			// Không blend tại bước chuyển hệ tọa độ.
			MotionBlendRadius := 0.0;
	
			// Motion chạy trong Robot Base/MCS.
			MotionCoordSystem := E_AppCoordSystem.APP_COORD_ROBOT_BASE;
	
			// MoveL.
			MotionCommand := 2;
	
			// Phát yêu cầu tới Motion Adapter.
			xMotionRequestPending := TRUE;
			xMotionIssued := TRUE;
	
		END_IF;
	
		// Motion Adapter đã nhận lệnh.
		IF MotionAccepted AND xMotionRequestPending THEN
			xMotionRequestPending := FALSE;
			xMotionActive := TRUE;
		END_IF;
	
		// Điểm Safe Leave hoàn thành.
		IF MotionDone AND xMotionActive THEN
	
			xMotionActive := FALSE;
			xMotionIssued := FALSE;
			xMotionRequestPending := FALSE;
	
			Runtime.State := E_TrackingState.TRK_MOVE_PLACE;
	
		// Motion Safe Leave báo lỗi.
		ELSIF MotionError AND xMotionActive THEN
	
			xMotionActive := FALSE;
			xMotionIssued := FALSE;
			xMotionRequestPending := FALSE;
	
			Runtime.Response.Error := TRUE;
			Runtime.Response.ErrorID := MotionErrorID;
	
			Runtime.State := E_TrackingState.TRK_ERROR;
	
		END_IF;
		

    //=========================================================================
    // TRK_MOVE_PLACE
    // Di chuyển từ LeavePos tới PlacePos trong hệ robot/base.
    //=========================================================================
    E_TrackingState.TRK_MOVE_PLACE:

        // Giữ hút tới khi tới điểm đặt.
        VacuumCommand := xVacuumCaptured;

        // Tạo request Place mới.
        IF NOT xMotionIssued AND NOT xMotionRequestPending AND NOT xMotionActive THEN

            // Gán điểm Place.
            MotionTarget := Config.PlacePos;

            // Gán tốc độ Place.
            MotionSpeed := Config.Motion.Place.Speed;

            // Gán gia tốc Place.
            MotionAcceleration := Config.Motion.Place.Acceleration;

            // Gán giảm tốc Place.
            MotionDeceleration := Config.Motion.Place.Deceleration;

            // Gán jerk Place.
            MotionJerk := Config.Motion.Place.Jerk;

            // Gán blend Place.
            MotionBlendRadius := Config.Motion.Place.BlendRadius;

            // Place chạy trong hệ robot/base.
            MotionCoordSystem := E_AppCoordSystem.APP_COORD_ROBOT_BASE;

            // Mã lệnh MoveL.
            MotionCommand := 2;

            // Bật request pending.
            xMotionRequestPending := TRUE;

            // Đánh dấu đã tạo lệnh.
            xMotionIssued := TRUE;
        END_IF;

        // Adapter đã nhận request.
        IF MotionAccepted AND xMotionRequestPending THEN
            xMotionRequestPending := FALSE;
            xMotionActive := TRUE;
        END_IF;

        // Place hoàn thành.
        IF MotionDone AND xMotionActive THEN
            xMotionActive := FALSE;
            xMotionIssued := FALSE;

            Runtime.State := E_TrackingState.TRK_RELEASE_PRODUCT;

        // Place lỗi.
        ELSIF MotionError AND xMotionActive THEN
            xMotionActive := FALSE;

            Runtime.Response.Error := TRUE;
            Runtime.Response.ErrorID := MotionErrorID;

            Runtime.State := E_TrackingState.TRK_ERROR;
        END_IF;

    //=========================================================================
    // TRK_RELEASE_PRODUCT
    // Tắt hút, bật thổi và chuẩn bị timer.
    //=========================================================================
    E_TrackingState.TRK_RELEASE_PRODUCT:

        // Tắt hút để nhả sản phẩm.
        VacuumCommand := FALSE;

        // Bật van thổi.
        BlowCommand := TRUE;

        // Reset timer thổi trước khi vào state chờ.
        tonBlow(IN := FALSE);

        // Chuyển sang chờ đủ thời gian thổi.
        Runtime.State := E_TrackingState.TRK_WAIT_BLOW;

    //=========================================================================
    // TRK_WAIT_BLOW
    // Giữ thổi trong Config.BlowTime.
    //=========================================================================
    E_TrackingState.TRK_WAIT_BLOW:

        // Bảo đảm hút tắt.
        VacuumCommand := FALSE;

        // Giữ van thổi bật.
        BlowCommand := TRUE;

        // Chạy timer thổi.
        tonBlow(
            IN := TRUE,
            PT := Config.BlowTime
        );

        // Khi hết thời gian thổi.
        IF tonBlow.Q THEN
            // Reset timer.
            tonBlow(IN := FALSE);

            // Tắt thổi.
            BlowCommand := FALSE;

            // Đánh dấu object đã PICKED.
            Queue.Objects[Runtime.SelectedObjectIndex].State := E_TrackingObjectState.OBJ_PICKED;

            // Giải phóng cờ Reserved.
            Queue.Objects[Runtime.SelectedObjectIndex].Reserved := FALSE;

            // Giải phóng ActiveIndex.
            Queue.ActiveIndex := GVL.C_INVALID_INDEX;

            // Báo gắp thành công.
            Runtime.PickSuccess := TRUE;

            // Xóa object active trong Runtime.
            Runtime.SelectedObjectIndex := 0;
            Runtime.SelectedObjectID := 0;

            // Xóa trạng thái đã giữ vật.
            xVacuumCaptured := FALSE;

            // Phát Done.
            Runtime.Response.Done := TRUE;

            // Chuyển sang Complete.
            Runtime.State := E_TrackingState.TRK_COMPLETE;
        END_IF;

    //=========================================================================
    // TRK_COMPLETE
    // Kết thúc một object; nếu Execute còn TRUE thì tìm object tiếp theo.
    //=========================================================================
    E_TrackingState.TRK_COMPLETE:

        // Chu trình một object đã hoàn thành.
		Runtime.Response.Busy := FALSE;
		Runtime.Response.Done := TRUE;
	
		// Giữ output ở trạng thái an toàn.
		VacuumCommand := FALSE;
		BlowCommand := FALSE;
	
		// Chỉ về IDLE khi tầng Command Engine hạ Execute.
		IF NOT Execute THEN
			Runtime.Response.Accepted := FALSE;
			Runtime.Response.Done := FALSE;
			Runtime.State := E_TrackingState.TRK_IDLE;
		END_IF;


    //=========================================================================
    // TRK_ABORT_ACTIVE
    // Hủy motion vì object vượt vùng trước khi VacuumOK.
    //=========================================================================
    E_TrackingState.TRK_ABORT_ACTIVE:

        // Tắt hút vì chưa giữ được vật.
        VacuumCommand := FALSE;

        // Tắt thổi.
        BlowCommand := FALSE;

        // Bật yêu cầu abort motion.
        MotionAbort := TRUE;

        // Khi Motion Manager xác nhận abort hoàn tất.
        IF MotionAbortDone THEN
            // Hạ yêu cầu abort.
            MotionAbort := FALSE;

            // Xóa trạng thái motion.
            xMotionIssued := FALSE;
            xMotionRequestPending := FALSE;
            xMotionActive := FALSE;

            // Nếu PCS không còn InUse thì có thể tắt tracking.
            IF NOT fbTrackBelt.InUse THEN
                xTrackExecute := FALSE;

                // Chuyển sang vị trí an toàn.
                Runtime.State := E_TrackingState.TRK_MOVE_SAFE;
            END_IF;
        END_IF;

    //=========================================================================
    // TRK_MOVE_SAFE
    // Đưa robot về LeavePos sau khi bỏ object.
    //=========================================================================
    E_TrackingState.TRK_MOVE_SAFE:

        // Tắt hút.
        VacuumCommand := FALSE;

        // Tạo request Move Safe.
        IF NOT xMotionIssued AND NOT xMotionRequestPending AND NOT xMotionActive THEN

            // Dùng LeavePos làm điểm an toàn.
            MotionTarget := Config.LeavePos;

            // Dùng thông số Leave.
            MotionSpeed := Config.Motion.Leave.Speed;

            MotionAcceleration := Config.Motion.Leave.Acceleration;

            MotionDeceleration := Config.Motion.Leave.Deceleration;

            MotionJerk := Config.Motion.Leave.Jerk;

            MotionBlendRadius := Config.Motion.Leave.BlendRadius;

            // Chạy trong hệ robot/base.
            MotionCoordSystem := E_AppCoordSystem.APP_COORD_ROBOT_BASE;

            // Mã lệnh MoveL.
            MotionCommand := 2;

            // Bật request pending.
            xMotionRequestPending := TRUE;

            // Đánh dấu đã tạo lệnh.
            xMotionIssued := TRUE;
        END_IF;

        // Adapter đã nhận request.
        IF MotionAccepted AND xMotionRequestPending THEN
            xMotionRequestPending := FALSE;
            xMotionActive := TRUE;
        END_IF;

        // Move Safe hoàn thành.
        IF MotionDone AND xMotionActive THEN
            xMotionActive := FALSE;
            xMotionIssued := FALSE;

            Runtime.State := E_TrackingState.TRK_RELEASE_OBJECT;

        // Move Safe lỗi.
        ELSIF MotionError AND xMotionActive THEN
            xMotionActive := FALSE;

            Runtime.Response.Error := TRUE;
            Runtime.Response.ErrorID := MotionErrorID;

            Runtime.State := E_TrackingState.TRK_ERROR;
        END_IF;

    //=========================================================================
    // TRK_RELEASE_OBJECT
    // Giải phóng object MISSED và tiếp tục object kế tiếp.
    //=========================================================================
    E_TrackingState.TRK_RELEASE_OBJECT:

        // Tắt hút.
        VacuumCommand := FALSE;

        // Chỉ release khi PCS không còn InUse.
        IF NOT fbTrackBelt.InUse THEN
            // Tắt tracking PCS.
            xTrackExecute := FALSE;

            // Kiểm tra index trước khi truy cập Queue.
            IF Runtime.SelectedObjectIndex >= 1 AND Runtime.SelectedObjectIndex <= GVL.C_MAX_TRACK_OBJECTS THEN

                // Giải phóng object.
                Queue.Objects[Runtime.SelectedObjectIndex].Reserved := FALSE;
            END_IF;

            // Giải phóng ActiveIndex.
            Queue.ActiveIndex := GVL.C_INVALID_INDEX;

            // Xóa object active trong Runtime.
            Runtime.SelectedObjectIndex := 0;
            Runtime.SelectedObjectID := 0;

            // Xóa thông tin PCS.
            Runtime.PCSInfo.Valid := FALSE;
            Runtime.PCSInfo.InUse := FALSE;

            // Xóa trạng thái tool.
            xVacuumCaptured := FALSE;

            // Xóa trạng thái motion.
            xMotionIssued := FALSE;
            xMotionRequestPending := FALSE;
            xMotionActive := FALSE;

            // Tiếp tục tìm object khác.
            Runtime.State := E_TrackingState.TRK_FIND_OBJECT;
        END_IF;

    //=========================================================================
    // TRK_ABORTING
    // Hủy toàn ứng dụng khi Execute bị hạ.
    //=========================================================================
    E_TrackingState.TRK_ABORTING:

        // Tắt hút.
        VacuumCommand := FALSE;

        // Tắt thổi.
        BlowCommand := FALSE;

        // Yêu cầu abort motion.
        MotionAbort := TRUE;

        // Nếu có object active thì đánh dấu ABORTED.
        IF Runtime.SelectedObjectIndex >= 1 AND Runtime.SelectedObjectIndex <= GVL.C_MAX_TRACK_OBJECTS THEN

            Queue.Objects[Runtime.SelectedObjectIndex].State := E_TrackingObjectState.OBJ_ABORTED;

            Queue.Objects[Runtime.SelectedObjectIndex].Reserved := FALSE;
        END_IF;

        // Khi abort motion xong và PCS không còn InUse.
        IF MotionAbortDone AND NOT fbTrackBelt.InUse THEN

            // Hạ abort.
            MotionAbort := FALSE;

            // Tắt tracking PCS.
            xTrackExecute := FALSE;

            // Giải phóng ActiveIndex.
            Queue.ActiveIndex := GVL.C_INVALID_INDEX;

            // Xóa object active.
            Runtime.SelectedObjectIndex := 0;
            Runtime.SelectedObjectID := 0;

            // Xóa Busy và Accepted.
            Runtime.Response.Busy := FALSE;
            Runtime.Response.Accepted := FALSE;

            // Về IDLE.
            Runtime.State := E_TrackingState.TRK_IDLE;
        END_IF;

    //=========================================================================
    // TRK_ERROR
    // Giữ lỗi để Application Manager/HMI đọc.
    //=========================================================================
    E_TrackingState.TRK_ERROR:

        // Manager không còn xử lý bình thường.
        Runtime.Response.Busy := FALSE;

        // Giữ cờ Error.
        Runtime.Response.Error := TRUE;

        // Tắt hút.
        VacuumCommand := FALSE;

        // Tắt thổi.
        BlowCommand := FALSE;

        // Yêu cầu abort motion.
        MotionAbort := TRUE;

        // Nếu có object active thì đánh dấu ERROR.
        IF Runtime.SelectedObjectIndex >= 1 AND Runtime.SelectedObjectIndex <= GVL.C_MAX_TRACK_OBJECTS THEN

            Queue.Objects[Runtime.SelectedObjectIndex].State := E_TrackingObjectState.OBJ_ERROR;

            Queue.Objects[Runtime.SelectedObjectIndex].Reserved := FALSE;
        END_IF;

        // Chỉ tắt tracking khi PCS không còn InUse.
        IF NOT fbTrackBelt.InUse THEN
            xTrackExecute := FALSE;
        END_IF;

    //=========================================================================
    // STATE KHÔNG HỢP LỆ
    //=========================================================================
    ELSE
        // Báo lỗi state không hợp lệ.
        Runtime.Response.Error := TRUE;

        // Mã lỗi nội bộ cho state không hợp lệ.
        Runtime.Response.ErrorID := 6999;

        // Chuyển về TRK_ERROR.
        Runtime.State := E_TrackingState.TRK_ERROR;

END_CASE;

END_FUNCTION_BLOCK

// Just_Motion_Control_x86_64_Linux_SM_WV/Application/FB_/ConveyorTrack/FB_TrackingMotionQueueAdapter_B
FUNCTION_BLOCK FB_TrackingMotionQueueAdapter_B
VAR_INPUT
    Enable : BOOL; // Biến nội bộ Enable.
    Reset : BOOL; // Biến nội bộ Reset.
    Request : BOOL; // Biến nội bộ Request.
    Abort : BOOL; // Biến nội bộ Abort.
    Target : ST_POS; // Biến nội bộ Target.
    Speed : REAL; // Biến nội bộ Speed.
    Acceleration : REAL; // Biến nội bộ Acceleration.
    Deceleration : REAL; // Biến nội bộ Deceleration.
    Jerk : REAL; // Biến nội bộ Jerk.
    BlendRadius : REAL; // Biến nội bộ BlendRadius.
    CoordSystem : E_AppCoordSystem; // Biến nội bộ CoordSystem.
    Command : UINT; // Biến nội bộ Command.
    LogicSimulation : BOOL; // Logic-only simulation không push vào robot.
    LogicMotionDuration : TIME := TIME#300ms; // Biến nội bộ LogicMotionDuration.
END_VAR

VAR_OUTPUT
    Accepted : BOOL; // Biến nội bộ Accepted.
    Busy : BOOL; // Biến nội bộ Busy.
    Done : BOOL; // Biến nội bộ Done.
    Error : BOOL; // Biến nội bộ Error.
    ErrorID : UDINT; // Biến nội bộ ErrorID.
    AbortDone : BOOL; // Biến nội bộ AbortDone.
END_VAR

VAR
    fbPush : FB_MotionQueuePush_B; // Biến nội bộ fbPush.
    rtRequest : R_TRIG; // Biến nội bộ rtRequest.
    tonLogicMotion : TON; // Biến nội bộ tonLogicMotion.
    stItem : ST_MotionQueueItem; // Biến nội bộ stItem.
    xPushExecute : BOOL; // Biến nội bộ xPushExecute.
    xWaitingMotionResult : BOOL; // Biến nội bộ xWaitingMotionResult.
    xAcceptedLatched : BOOL; // Biến nội bộ xAcceptedLatched.
    diRequestSequence : DINT := -1000; // Biến nội bộ diRequestSequence.
    iActiveSourceStep : INT; // Biến nội bộ iActiveSourceStep.
END_VAR

Accepted := FALSE;
Done := FALSE;
AbortDone := FALSE;

// Error không nên giữ từ request cũ khi Adapter đang không chờ motion.
IF NOT xPushExecute AND NOT xWaitingMotionResult THEN
    Error := FALSE;
    ErrorID := 0;
END_IF;

// IF Reset OR NOT Enable THEN
//     xPushExecute := FALSE;
//     xWaitingMotionResult := FALSE;
//     xAcceptedLatched := FALSE;
//     Busy := FALSE;
//     Error := FALSE;
//     ErrorID := 0;
//     tonLogicMotion(IN := FALSE);
//     fbPush(Execute := FALSE, Item := stItem);
//     RETURN;
// END_IF;

IF Reset OR NOT Enable THEN

    // Hạ yêu cầu push vào Motion Queue.
    xPushExecute := FALSE;

    // Không còn chờ kết quả motion trước.
    xWaitingMotionResult := FALSE;

    // Xóa cờ Accepted nội bộ.
    xAcceptedLatched := FALSE;

    // Xóa trạng thái output.
    Accepted := FALSE;
    Busy := FALSE;
    Done := FALSE;
    Error := FALSE;
    ErrorID := 0;
    AbortDone := FALSE;

    // Xóa SourceStep của request cũ.
    iActiveSourceStep := 0;

    // Hạ yêu cầu Abort còn sót lại.
    GVL.B_MotionAbortReq := FALSE;

    // Reset timer mô phỏng.
    tonLogicMotion(IN := FALSE);

    // Reset FB Push Motion Queue.
    fbPush(Execute := FALSE, Item := stItem);

    RETURN;
END_IF;

IF Abort THEN
    IF LogicSimulation THEN
        xWaitingMotionResult := FALSE;
        Busy := FALSE;
        AbortDone := TRUE;
    ELSE
        GVL.B_MotionAbortReq := TRUE;
        IF GVL.B_MotionAbortDone THEN
            GVL.B_MotionAbortReq := FALSE;
            xWaitingMotionResult := FALSE;
            Busy := FALSE;
            AbortDone := TRUE;
        END_IF;
    END_IF;
    RETURN;
END_IF;

rtRequest(CLK := Request);

//=============================================================================
// LOGIC-ONLY SIMULATION
//=============================================================================
IF LogicSimulation THEN
    IF rtRequest.Q AND NOT Busy THEN
        Accepted := TRUE;
        Busy := TRUE;
        tonLogicMotion(IN := FALSE);
    END_IF;

    tonLogicMotion(IN := Busy, PT := LogicMotionDuration);

    IF tonLogicMotion.Q THEN
        tonLogicMotion(IN := FALSE);
        Busy := FALSE;
        Done := TRUE;
    END_IF;

    RETURN;
END_IF;

//=============================================================================
// ROBOT REAL: ĐÓNG GÓI VÀ PUSH VÀO MOTION QUEUE ROBOT B
//=============================================================================
IF rtRequest.Q AND NOT xPushExecute AND NOT xWaitingMotionResult THEN
    diRequestSequence := diRequestSequence - 1;
    IF diRequestSequence < -30000 THEN diRequestSequence := -1000; END_IF;
    iActiveSourceStep := DINT_TO_INT(diRequestSequence);

    stItem.Cmd := E_RobotCmd.CMD_MovL;
    stItem.SourceStep := iActiveSourceStep;
    stItem.PointNo := 0;
    stItem.MidPointNo := 0;
    stItem.EndPointNo := 0;
    stItem.Speed := REAL_TO_LREAL(Speed);
    stItem.BlendMode := GVL.C_TM_None;
    stItem.BlendRadius := REAL_TO_LREAL(BlendRadius);
    stItem.CircleMode := 0;
    stItem.PathChoice := 0;
    stItem.SkipPositionCheck := TRUE;

    stItem.UseDirectPosition := TRUE;
    stItem.DirectPosition := Target;
    stItem.DirectCoordSystem := F_MapAppCoordSystem(Coord := CoordSystem);
    stItem.Acceleration := REAL_TO_LREAL(Acceleration);
    stItem.Deceleration := REAL_TO_LREAL(Deceleration);
    stItem.Jerk := REAL_TO_LREAL(Jerk);
    stItem.ApplicationCommandID := TO_UDINT(ABS(iActiveSourceStep));

    xPushExecute := TRUE;
END_IF;

fbPush(Execute := xPushExecute, Item := stItem);

IF xPushExecute AND fbPush.Done THEN
    xPushExecute := FALSE;
    xWaitingMotionResult := TRUE;
    xAcceptedLatched := TRUE;
    Accepted := TRUE;
    Busy := TRUE;
END_IF;

IF xPushExecute AND fbPush.Error THEN
    xPushExecute := FALSE;
    Error := TRUE;
    ErrorID := 7201; // Motion Queue full / Push failed.
END_IF;

// Reset handshake của FB Push sau khi push xong.
IF NOT xPushExecute THEN fbPush(Execute := FALSE, Item := stItem); END_IF;

// Theo dõi đúng item bằng SourceStep âm riêng của Application.
IF xWaitingMotionResult THEN
    Busy := TRUE;

//     IF GVL.B_MotionDonePulse AND GVL.B_MotionDoneStep = iActiveSourceStep THEN
//         xWaitingMotionResult := FALSE;
//         Busy := FALSE;
//         Done := TRUE;
//     END_IF;
// 
//     IF GVL.B_MotionErrorPulse AND GVL.B_MotionErrorStep = iActiveSourceStep THEN
//         xWaitingMotionResult := FALSE;
//         Busy := FALSE;
//         Error := TRUE;
//         ErrorID := INT_TO_UDINT(GVL.B_MotionErrorCode);
//     END_IF;
	
	IF GVL.B_MotionDonePulse AND GVL.B_MotionDoneStep = iActiveSourceStep THEN
		xWaitingMotionResult := FALSE;
		xAcceptedLatched := FALSE;
		Busy := FALSE;
		Done := TRUE;
	END_IF;
	
	// Motion hiện tại báo lỗi đúng SourceStep.
	IF GVL.B_MotionErrorPulse AND GVL.B_MotionErrorStep = iActiveSourceStep THEN
		xWaitingMotionResult := FALSE;
		xAcceptedLatched := FALSE;
		Busy := FALSE;
		Error := TRUE;
		ErrorID := INT_TO_UDINT(GVL.B_MotionErrorCode);
	END_IF;
END_IF;

END_FUNCTION_BLOCK

// Just_Motion_Control_x86_64_Linux_SM_WV/Application/FB_/TOOL/FB_SelectRobotTool_B
FUNCTION_BLOCK FB_SelectRobotTool_B
VAR_INPUT
    Execute : BOOL; // Xung Execute.
    Reset : BOOL; // Reset FB.
    ToolID : UINT; // ToolID cần chọn.
END_VAR

VAR_OUTPUT
    Done : BOOL; // Tool đã được chọn.
    Busy : BOOL; // FB đang xử lý.
    Error : BOOL; // FB lỗi.
    ErrorID : UDINT; // Mã lỗi.
END_VAR

VAR
    rtExecute : R_TRIG; // Bắt cạnh Execute.
    fbGroupSetTool : SMC_GroupSetTool; // TODO: Khai báo instance SMC_GroupSetTool đúng theo version thư viện.
    xExecuteTool : BOOL; // Biến nội bộ xExecuteTool.
    udiMyRequestID : UDINT := 0; // RequestID thuộc transaction hiện tại.
END_VAR

//=============================================================================
// FB_SelectRobotTool
//-----------------------------------------------------------------------------
// ToolID = Number_Tool.
// Không gọi SMC_GroupSetTool tại đây.
// POU_COORDINATE_ là nơi duy nhất Apply TCP vào SCARA_B.
//=============================================================================

Done := FALSE;


//=============================================================================
// RESET
//=============================================================================
IF Reset THEN
    Busy := FALSE;
    Error := FALSE;
    ErrorID := 0;
    udiMyRequestID := 0;
    RETURN;
END_IF;


//=============================================================================
// DETECT EXECUTE
//=============================================================================
rtExecute(CLK := Execute);


//=============================================================================
// TẠO YÊU CẦU CHỌN / APPLY TOOL
//=============================================================================
IF rtExecute.Q AND NOT Busy THEN

    Busy := TRUE;
    Error := FALSE;
    ErrorID := 0;

    //---------------------------------------------------------------------
    // ToolID chính là Number_Tool.
    //
    // ToolID = 0 : No Tool Offset.
    // ToolID = 1 : Tool 1.
    // ToolID = 2 : Tool 2...
    //---------------------------------------------------------------------
    GVL.RB_B.Number_Tool := ToolID;

    //---------------------------------------------------------------------
    // Luôn tạo Request mới.
    // Nhờ vậy cùng ToolID nhưng TCP đã thay đổi vẫn được Apply lại.
    //---------------------------------------------------------------------
    GVL.g_udiRobotBToolApplyRequestB := GVL.g_udiRobotBToolApplyRequestB + 1;
    IF GVL.g_udiRobotBToolApplyRequestB = 0 THEN GVL.g_udiRobotBToolApplyRequestB := 1; END_IF;

    // Chốt Request của transaction này.
    udiMyRequestID := GVL.g_udiRobotBToolApplyRequestB;

END_IF;


//=============================================================================
// CHỜ KẾT QUẢ TỪ POU_COORDINATE_
//=============================================================================
IF Busy THEN

    //---------------------------------------------------------------------
    // APPLY ERROR
    //---------------------------------------------------------------------
    IF GVL.g_xRobotBToolApplyError THEN
        Busy := FALSE;
        Error := TRUE;
        ErrorID := GVL.g_udiRobotBToolApplyErrorID;

    //---------------------------------------------------------------------
    // APPLY DONE
    //---------------------------------------------------------------------
    ELSIF udiMyRequestID <> 0
    AND GVL.g_udiRobotBToolAppliedRequestB = udiMyRequestID THEN
        Busy := FALSE;
        Error := FALSE;
        ErrorID := 0;
        Done := TRUE;
    END_IF;

END_IF;





// (*
// ===============================================================================
// FUNCTION BLOCK
//     FB_SelectRobotTool
// 
// DESCRIPTION
//     Wrapper chọn Tool/TCP cho Robot.
// 
// TODO INTEGRATIONđ
//     Thay phần Logic-Only Placeholder bằng SMC_GroupSetTool đang có
//     trong project hiện tại.
// 
// EXPECTED FLOW
//     Execute rising edge
//         -> Call SMC_GroupSetTool
//         -> Wait Done/Error
//         -> Return Done/Error
// ===============================================================================
// *)
// 
// //=============================================================================
// // DEFAULT PULSE OUTPUT
// //=============================================================================
// Done := FALSE;
// 
// 
// //=============================================================================
// // RESET
// //=============================================================================
// IF Reset THEN
// 
//     Busy := FALSE;
// 
//     Error := FALSE;
//     ErrorID := 0;
// 
//     RETURN;
// 
// END_IF;
// 
// 
// //=============================================================================
// // DETECT EXECUTE
// //=============================================================================
// rtExecute(CLK := Execute);
// 
// 
// //=============================================================================
// // START TOOL SELECTION
// //=============================================================================
// IF rtExecute.Q AND NOT Busy THEN
// 
//     Busy := TRUE;
// 
//     Error := FALSE;
//     ErrorID := 0;
// 
// 
//     //=========================================================================
//     // TODO: CALL SMC_GROUPSETTOOL HERE
//     //-------------------------------------------------------------------------
//     // Ví dụ logic:
//     //
// 	fbGroupSetTool(
// 		Execute   := TRUE,
// 		AxisGroup := SCARA_B,
// 		ToolOffset := F_ConvertToolTCP(ToolTCP)
// 	);
// 	
// 	IF fbGroupSetTool.Done THEN
// 		Busy := FALSE;
// 		Done := TRUE;
// 	END_IF;
// 	
// 	IF fbGroupSetTool.Error THEN
// 		Busy := FALSE;
// 		Error := TRUE;
// 		ErrorID := fbGroupSetTool.ErrorID;
// 	END_IF;
//     //=========================================================================
// 
// 
// //     //-------------------------------------------------------------------------
// //     // LOGIC-ONLY PLACEHOLDER
// //     //-------------------------------------------------------------------------
// //     // Xóa hai dòng dưới sau khi nối SMC_GroupSetTool thực tế.
// //     Busy := FALSE;
// //     Done := TRUE;
// 
// END_IF;

END_FUNCTION_BLOCK

// Just_Motion_Control_x86_64_Linux_SM_WV/Application/FB_/TOOL/FB_ToolManager_B
FUNCTION_BLOCK FB_ToolManager_B
VAR_INPUT
    Enable : BOOL; // Cho phép Tool Manager.
    Command : ST_ToolCommand; // Command hiện tại.
    Config : ST_ToolConfig; // Cấu hình Tool.
END_VAR

VAR_IN_OUT
    Status : ST_ToolStatus; // Runtime Status của Tool.
END_VAR

VAR
    rtExecute : R_TRIG; // Bắt cạnh lên của Execute.
    eActiveCommand : E_ToolCommandType; // Lệnh Tool đang chạy.
    tonAction : TON; // Timer dùng khi không cấu hình DI.
    tonTimeout : TON; // Timer giới hạn thời gian lệnh Tool.
    tonConfirm : TON; // Timer xác nhận GripOK ổn định.
    xActionOK : BOOL; // Điều kiện lệnh Tool hoàn thành.
    xFeedbackDI : BOOL; // Giá trị DI đang kiểm tra.
    tAction : TIME; // Thời gian giả lập nếu không có Sensor.
    tTimeout : TIME; // Timeout của lệnh Tool.
END_VAR

(*
===============================================================================
FUNCTION BLOCK
    FB_ToolManager

DESCRIPTION
    Điều khiển một Tool độc lập.

SUPPORTED COMMANDS
    - DOWN
    - GRIP
    - UP
    - RELEASE

FEEDBACK RULE
    - Nếu DI Channel > 0:
          Dùng DI làm điều kiện hoàn thành.
    - Nếu DI Channel = 0:
          Dùng Timer cấu hình tương ứng.
    - Nếu UseUpDown = FALSE:
          DOWN và UP hoàn thành ngay.

IMPORTANT
    - Chỉ FB này được phép ghi request IO của Tool.
    - Interpreter không nên ghi trực tiếp vào các DO đã thuộc Tool.
===============================================================================
*)

//=============================================================================
// DEFAULT PULSE OUTPUTS
//=============================================================================
Status.Accepted := FALSE;
Status.Done := FALSE;


//=============================================================================
// COPY TOOL ID TO STATUS
//=============================================================================
Status.ToolID := Config.ToolID;


//=============================================================================
// RESET / DISABLE
//=============================================================================
IF NOT Enable OR Command.Reset THEN

    Status.Busy := FALSE;

    Status.Error := FALSE;
    Status.ErrorID := 0;

    Status.State :=
        E_ToolRuntimeState.IDLE;

    tonAction(IN := FALSE);
    tonTimeout(IN := FALSE);
    tonConfirm(IN := FALSE);

    RETURN;

END_IF;


//=============================================================================
// ABORT
//=============================================================================
IF Command.Abort THEN

    Status.Busy := FALSE;

    Status.Error := TRUE;
    Status.ErrorID := 9299;

    Status.State :=
        E_ToolRuntimeState.ERROR;

    RETURN;

END_IF;


//=============================================================================
// DETECT NEW COMMAND
//=============================================================================
rtExecute(CLK := Command.Execute);

IF rtExecute.Q AND NOT Status.Busy THEN

    // Lưu loại lệnh hiện tại.
    eActiveCommand :=
        Command.CommandType;

    // Handshake.
    Status.Accepted := TRUE;
    Status.Busy := TRUE;

    Status.Error := FALSE;
    Status.ErrorID := 0;

    Status.ResponseCommandID :=
        Command.CommandID;

    // Reset timer trước khi bắt đầu lệnh mới.
    tonAction(IN := FALSE);
    tonTimeout(IN := FALSE);
    tonConfirm(IN := FALSE);

    // Gán State runtime.
    CASE eActiveCommand OF

        E_ToolCommandType.DOWN:
            Status.State :=
                E_ToolRuntimeState.DOWNING;

        E_ToolCommandType.GRIP:
            Status.State :=
                E_ToolRuntimeState.GRIPPING;

        E_ToolCommandType.UP:
            Status.State :=
                E_ToolRuntimeState.UPPING;

        E_ToolCommandType.RELEASE:
            Status.State :=
                E_ToolRuntimeState.RELEASING;

        ELSE
            Status.Busy := FALSE;
            Status.Done := TRUE;

    END_CASE;

END_IF;


//=============================================================================
// NO ACTIVE COMMAND
//=============================================================================
IF NOT Status.Busy THEN
    RETURN;
END_IF;


//=============================================================================
// RESET LOCAL ACTION FLAGS
//=============================================================================
xActionOK := FALSE;
xFeedbackDI := FALSE;

tAction := T#0MS;
tTimeout := T#1S;


//=============================================================================
// EXECUTE ACTIVE COMMAND
//=============================================================================
CASE eActiveCommand OF


    //=========================================================================
    // ACTION: DOWN
    //=========================================================================
    E_ToolCommandType.DOWN:

        // Tool không có cơ cấu Up/Down.
        IF NOT Config.UseUpDown THEN

            xActionOK := TRUE;

        ELSE

            //-----------------------------------------------------------------
            // COMMAND DOWN OUTPUT
            //-----------------------------------------------------------------
			
			IF Config.IO.UseSingleUpDownDO THEN
				// Single DO: phat muc DOWN.
				IF Config.IO.UpDownDOChannel > 0 AND Config.IO.UpDownDOChannel <= GVL.C_MAX_DO THEN
					GVL.Y[Config.IO.UpDownDOChannel] := Config.IO.DownDOActiveLevel;
				END_IF;
			ELSE
				// Dual DO: bat Down, tat Up.
				IF Config.IO.DownDOChannel > 0 AND Config.IO.DownDOChannel <= GVL.C_MAX_DO THEN
					GVL.Y[Config.IO.DownDOChannel] := Config.IO.DownDOActiveLevel;
				END_IF;
			
				IF Config.IO.UpDOChannel > 0 AND Config.IO.UpDOChannel <= GVL.C_MAX_DO THEN
					GVL.Y[Config.IO.UpDOChannel] := NOT Config.IO.UpDOActiveLevel;
				END_IF;
			END_IF;


            //-----------------------------------------------------------------
            // CHECK DOWN FEEDBACK
            //-----------------------------------------------------------------
            IF Config.IO.DownOKDIChannel = 0 THEN

                // Không có DI -> dùng Timer.
                tAction :=
                    Config.DownTimeNoSensor;

                tonAction(
                    IN := TRUE,
                    PT := tAction
                );

                xActionOK :=
                    tonAction.Q;

            ELSE

                // Có DI -> dùng Sensor.
                xActionOK :=
                    GVL.X[
                        Config.IO.DownOKDIChannel
                    ] = Config.IO.DownOKDIActiveLevel;

            END_IF;


            // Timeout của DOWN.
            tTimeout :=
                Config.DownTimeout;

        END_IF;


    //=========================================================================
    // ACTION: GRIP
    //=========================================================================
    E_ToolCommandType.GRIP:

        //---------------------------------------------------------------------
        // RESET RELEASE OUTPUT
        //---------------------------------------------------------------------
        IF Config.IO.UseSingleGripReleaseDO THEN
			IF Config.IO.GripReleaseDOChannel > 0 AND Config.IO.GripReleaseDOChannel <= GVL.C_MAX_DO THEN
				GVL.Y[Config.IO.GripReleaseDOChannel] := Config.IO.GripDOActiveLevel;
			END_IF;
		ELSE
			IF Config.IO.ReleaseDOChannel > 0 AND Config.IO.ReleaseDOChannel <= GVL.C_MAX_DO THEN
				GVL.Y[Config.IO.ReleaseDOChannel] := NOT Config.IO.ReleaseDOActiveLevel;
			END_IF;
			IF Config.IO.GripDOChannel > 0 AND Config.IO.GripDOChannel <= GVL.C_MAX_DO THEN
				GVL.Y[Config.IO.GripDOChannel] := Config.IO.GripDOActiveLevel;
			END_IF;
		END_IF;


        //---------------------------------------------------------------------
        // CHECK GRIP FEEDBACK
        //---------------------------------------------------------------------
        IF Config.IO.GripOKDIChannel = 0 THEN

            // Không có GripOK DI -> dùng Timer.
            tAction :=
                Config.GripTimeNoSensor;

            tonAction(
                IN := TRUE,
                PT := tAction
            );

            xActionOK :=
                tonAction.Q;

        ELSE

            // Có GripOK DI.
            xFeedbackDI :=
                GVL.X[
                    Config.IO.GripOKDIChannel
                ] = Config.IO.GripOKDIActiveLevel;

            // Xác nhận tín hiệu ổn định.
            tonConfirm(
                IN := xFeedbackDI,
                PT := Config.GripConfirmDelay
            );

            xActionOK :=
                tonConfirm.Q;

        END_IF;


        // Timeout của GRIP.
        tTimeout :=
            Config.GripTimeout;


    //=========================================================================
    // ACTION: UP
    //=========================================================================
    E_ToolCommandType.UP:

        // Tool không có cơ cấu Up/Down.
        IF NOT Config.UseUpDown THEN

            xActionOK := TRUE;

        ELSE

            //-----------------------------------------------------------------
            // RESET DOWN OUTPUT
            //-----------------------------------------------------------------
			IF Config.IO.UseSingleUpDownDO THEN
				// Single DO: UP = dao muc DOWN.
				IF Config.IO.UpDownDOChannel > 0 AND Config.IO.UpDownDOChannel <= GVL.C_MAX_DO THEN
					GVL.Y[Config.IO.UpDownDOChannel] := NOT Config.IO.DownDOActiveLevel;
				END_IF;
			ELSE
				// Dual DO: tat Down, bat Up.
				IF Config.IO.DownDOChannel > 0 AND Config.IO.DownDOChannel <= GVL.C_MAX_DO THEN
					GVL.Y[Config.IO.DownDOChannel] := NOT Config.IO.DownDOActiveLevel;
				END_IF;
			
				IF Config.IO.UpDOChannel > 0 AND Config.IO.UpDOChannel <= GVL.C_MAX_DO THEN
					GVL.Y[Config.IO.UpDOChannel] := Config.IO.UpDOActiveLevel;
				END_IF;
			END_IF;


            //-----------------------------------------------------------------
            // CHECK UP FEEDBACK
            //-----------------------------------------------------------------
            IF Config.IO.UpOKDIChannel = 0 THEN

                // Không có DI -> dùng Timer.
                tAction :=
                    Config.UpTimeNoSensor;

                tonAction(
                    IN := TRUE,
                    PT := tAction
                );

                xActionOK :=
                    tonAction.Q;

            ELSE

                // Có DI -> dùng Sensor.
                xActionOK :=
                    GVL.X[
                        Config.IO.UpOKDIChannel
                    ] = Config.IO.UpOKDIActiveLevel;

            END_IF;


            // Timeout của UP.
            tTimeout :=
                Config.UpTimeout;

        END_IF;


    //=========================================================================
    // ACTION: RELEASE
    //=========================================================================
    E_ToolCommandType.RELEASE:

        //---------------------------------------------------------------------
        // RESET GRIP OUTPUT
        //---------------------------------------------------------------------
        IF Config.IO.UseSingleGripReleaseDO THEN
			IF Config.IO.GripReleaseDOChannel > 0 AND Config.IO.GripReleaseDOChannel <= GVL.C_MAX_DO THEN
				GVL.Y[Config.IO.GripReleaseDOChannel] := NOT Config.IO.GripDOActiveLevel;
			END_IF;
		ELSE
			IF Config.IO.GripDOChannel > 0 AND Config.IO.GripDOChannel <= GVL.C_MAX_DO THEN
				GVL.Y[Config.IO.GripDOChannel] := NOT Config.IO.GripDOActiveLevel;
			END_IF;
			IF Config.IO.ReleaseDOChannel > 0 AND Config.IO.ReleaseDOChannel <= GVL.C_MAX_DO THEN
				GVL.Y[Config.IO.ReleaseDOChannel] := Config.IO.ReleaseDOActiveLevel;
			END_IF;
		END_IF;


        //---------------------------------------------------------------------
        // RELEASE CURRENTLY USES TIMER
        //---------------------------------------------------------------------
        tAction :=
            Config.ReleaseTimeNoSensor;

        tonAction(
            IN := TRUE,
            PT := tAction
        );

        xActionOK :=
            tonAction.Q;


        // Timeout của RELEASE.
        tTimeout :=
            Config.ReleaseTimeout;

END_CASE;


//=============================================================================
// ACTION TIMEOUT
//=============================================================================
tonTimeout(
    IN := TRUE,
    PT := tTimeout
);


//=============================================================================
// COMMAND COMPLETE
//=============================================================================
IF xActionOK THEN

    // Reset timer.
    tonAction(IN := FALSE);
    tonTimeout(IN := FALSE);
    tonConfirm(IN := FALSE);

    // Hoàn thành Handshake.
    Status.Busy := FALSE;
    Status.Done := TRUE;

    Status.Error := FALSE;
    Status.ErrorID := 0;


    //-------------------------------------------------------------------------
    // UPDATE TOOL RUNTIME STATE
    //-------------------------------------------------------------------------
    CASE eActiveCommand OF

        E_ToolCommandType.DOWN:

            Status.State :=
                E_ToolRuntimeState.DOWN;


        E_ToolCommandType.GRIP:

            Status.State :=
                E_ToolRuntimeState.OCCUPIED;

            Status.Occupied :=
                TRUE;

            Status.HeldObjectID :=
                Command.ObjectID;

            Status.GripOK :=
                TRUE;


        E_ToolCommandType.UP:

            IF Status.Occupied THEN

                Status.State :=
                    E_ToolRuntimeState.OCCUPIED;

            ELSE

                Status.State :=
                    E_ToolRuntimeState.UP;

            END_IF;


        E_ToolCommandType.RELEASE:

            Status.State :=
                E_ToolRuntimeState.IDLE;

            Status.Occupied :=
                FALSE;

            Status.HeldObjectID :=
                0;

            Status.GripOK :=
                FALSE;

    END_CASE;


//=============================================================================
// COMMAND ERROR
//=============================================================================
ELSIF tonTimeout.Q THEN

    Status.Busy := FALSE;

    Status.Error := TRUE;

    // Mã lỗi được tạo từ loại lệnh Tool.
    Status.ErrorID :=
        9200 + TO_UDINT(eActiveCommand);

    Status.State :=
        E_ToolRuntimeState.ERROR;

END_IF;

END_FUNCTION_BLOCK

// Just_Motion_Control_x86_64_Linux_SM_WV/Application/PRG_MACHINE/POU_MODBUS
PROGRAM POU_MODBUS
VAR
	
	Modbus_TCP_slave_0: JMCMB.modbusTCPslaveINI;
	slaveRegisters_0: JMCMB.slaveRegisters;
	DATA : ARRAY[0..2000] OF INT;
	id, id2, id3 : INT;
	
	Modbus_TCP_slave_1: JMCMB.modbusTCPslaveINI;
	slaveRegisters_1: JMCMB.slaveRegisters;
	DATA1 : ARRAY[0..2000] OF INT;
	uiCamera : UINT;
	iCameraBase : INT;
	Enable_Modbus_Camera : ARRAY[0..GVL.C_MAX_VISION_CHANNELS] OF BOOL;
END_VAR

ACT_TCP_Sever();
//ACT_modbus();

ACTION ACT_TCP_Sever:
Modbus_TCP_slave_0(en := TRUE,
					iniID := 1,
					port	:= 1010,
					TCP_UDP	:= 	0,
					DelayRespTime := 300,
					connected =>,
					errID =>,
					Info	=>,
					errTotal =>);
slaveRegisters_0(	iniID := 1,
					modeTCP_RTU := 0,
					startAddr := 0,
					total		:= 2000,
					trans_data	:= DATA,
					errId =>,
					Info	=>,
					CMDTimes	=>);
					

//Enable_Modbus_Camera[1] := TRUE;
FOR uiCamera := 1 TO GVL.C_MAX_VISION_CHANNELS DO
	IF (GVL.g_aVisionConfig[uiCamera].Enable) THEN
		iCameraBase := (UINT_TO_INT(uiCamera) - 1) * 300;
	
		// Robot -> Vision: chỉ ghi 100 register đầu của Camera.
		FOR id := 0 TO 99 DO
			DATA[iCameraBase + id] := TO_INT(GVL.MODBUS[iCameraBase + id]);
		END_FOR;
	
		// Vision -> Robot: chỉ đọc 200 register sau của Camera.
		FOR id2 := 100 TO 299 DO
			GVL.MODBUS[iCameraBase + id2] := TO_WORD(DATA[iCameraBase + id2]);
		END_FOR;
	END_IF;
END_FOR;

// User Modbus
FOR id := 1200 TO 1599 DO
	DATA[id] := TO_INT(GVL.MODBUS[id]);
END_FOR;

// Vision -> Robot: chỉ đọc 200 register sau của Camera.
FOR id2 := 1600 TO 1999 DO
	GVL.MODBUS[id2] := TO_WORD(DATA[id2]);
END_FOR;

// iCameraBase := 0;
// 	
// // Robot -> Vision: chỉ ghi 100 register đầu của Camera.
// FOR id := 0 TO 99 DO
// 	DATA[iCameraBase + id] := TO_INT(GVL.MODBUS[iCameraBase + id]);
// END_FOR;
// 
// // Vision -> Robot: chỉ đọc 200 register sau của Camera.
// FOR id2 := 100 TO 299 DO
// 	GVL.MODBUS[iCameraBase + id2] := TO_WORD(DATA[iCameraBase + id2]);
// END_FOR;
// 
// FOR id3 := 1500 TO 1999 DO
// 	GVL.MODBUS[id3] := TO_WORD(DATA[id3]);   // luôn cập nhật
// END_FOR;


Modbus_TCP_slave_1(en := FALSE,
					iniID := 2,
					port	:= 1012,
					TCP_UDP	:= 	0,
					DelayRespTime := 300,
					connected =>,
					errID =>,
					Info	=>,
					errTotal =>);
slaveRegisters_1(	iniID := 2,
					modeTCP_RTU := 0,
					startAddr := 0,
					total		:= 2000,
					trans_data	:= DATA1,
					errId =>,
					Info	=>,
					CMDTimes	=>);
END_ACTION

END_PROGRAM

// Just_Motion_Control_x86_64_Linux_SM_WV/Application/PRG_MACHINE/PRG_VisionConfigInit
PROGRAM PRG_VisionConfigInit
VAR
    xInitialized : BOOL := FALSE;
END_VAR

//=============================================================================
// PRG_VisionConfigInit
//-----------------------------------------------------------------------------
// Khởi tạo cấu hình Vision một lần sau khi PLC RUN.
// Không ghi lặp mỗi scan để sau này HMI có thể sửa cấu hình.
//=============================================================================

IF NOT xInitialized THEN

    //=========================================================================
    // CAMERA 1
    //=========================================================================
    //GVL.g_aVisionConfig[1].Enable := TRUE;
    GVL.g_aVisionConfig[1].CameraID := 1;
    GVL.g_aVisionConfig[1].BaseAddress := 0;
    GVL.g_aVisionConfig[1].CommandOffset := 0;
    GVL.g_aVisionConfig[1].StatusOffset := 100;
    GVL.g_aVisionConfig[1].HeaderOffset := 101;
    GVL.g_aVisionConfig[1].DataOffset := 116;

    // Scale tạm dùng cho test.
    // Raw 10000 -> 10.000 mm.
    //GVL.g_aVisionConfig[1].PositionScale := 0.001;
    //GVL.g_aVisionConfig[1].AngleScale := 0.001;
    GVL.g_aVisionConfig[1].ScoreScale := 1.0;

//     GVL.g_aVisionConfig[1].TriggerTimeout := T#2S;
//     GVL.g_aVisionConfig[1].ResultTimeout := T#3S;
    GVL.g_aVisionConfig[1].BlockTimeout := T#1S;
//     GVL.g_aVisionConfig[1].MaxPointCount := 12;
    //GVL.g_aVisionConfig[1].MaxRetry := 2;

	
	//=============================================================================
	// VISION TRACKING SOURCE 1
	//-----------------------------------------------------------------------------
	// Nguồn Vision dùng để tạo Object cho Conveyor Tracking Robot A.
	// CameraID và JobID phải khớp Header của Result.
	//=============================================================================
	
// 	GVL.g_aVisionTrackingSourceConfigA[1].Enable := TRUE;
// 	GVL.g_aVisionTrackingSourceConfigA[1].VisionSourceID := 1;
// 	GVL.g_aVisionTrackingSourceConfigA[1].VisionSourceName := 'Vision Tracking Cam 1';
// 	
// 	GVL.g_aVisionTrackingSourceConfigA[1].CameraID := 1;
// 	GVL.g_aVisionTrackingSourceConfigA[1].JobID := 1;
// 	
// 	// Nếu Vision không trả ProductClassID thì dùng Class mặc định này.
// 	GVL.g_aVisionTrackingSourceConfigA[1].ProductClassID := 1;
// 	
// 	// Chỉ nhận Object đạt Score yêu cầu.
// 	GVL.g_aVisionTrackingSourceConfigA[1].MinimumScore := 70.0;
// 	GVL.g_aVisionTrackingSourceConfigA[1].MaxObjectCount := 10;
	
	//=============================================================================
	// SCALE
	//-----------------------------------------------------------------------------
	// Result Modbus Driver hiện đã decode X/Y/A ra engineering unit,
	// vì vậy ResultInPixel phải FALSE trong bài test hiện tại.
	//=============================================================================
// 	GVL.g_aVisionTrackingSourceConfigA[1].ResultInPixel := FALSE;
// 	GVL.g_aVisionTrackingSourceConfigA[1].MMPerPixelX := 1.0;
// 	GVL.g_aVisionTrackingSourceConfigA[1].MMPerPixelY := 1.0;
// 	
// 	//=============================================================================
// 	// VISION FINE OFFSET
// 	//=============================================================================
// 	GVL.g_aVisionTrackingSourceConfigA[1].VisionOffset.X := 0.0;
// 	GVL.g_aVisionTrackingSourceConfigA[1].VisionOffset.Y := 0.0;
// 	GVL.g_aVisionTrackingSourceConfigA[1].VisionOffset.Z := 0.0;
// 	GVL.g_aVisionTrackingSourceConfigA[1].VisionOffset.A := 0.0;
	
// 	//=============================================================================
// 	// DUPLICATE FILTER
// 	//=============================================================================
// 	GVL.g_aVisionTrackingSourceConfigA[1].DuplicateToleranceXMM := 10.0;
// 	GVL.g_aVisionTrackingSourceConfigA[1].DuplicateToleranceYMM := 10.0;
// 	GVL.g_aVisionTrackingSourceConfigA[1].DuplicateAngleDeg := 5.0;
	
	//=============================================================================
	// BACKGROUND TRIGGER
	//-----------------------------------------------------------------------------
	// Trong lúc test dữ liệu giả lập, chưa bật AutoTrigger để tránh sinh TriggerID mới.
	//=============================================================================
// 	GVL.g_aVisionTrackingSourceConfigA[1].AutoTrigger := FALSE;
// 	GVL.g_aVisionTrackingSourceConfigA[1].TriggerPitchMM := 50.0;
// 	GVL.g_aVisionTrackingSourceConfigA[1].TriggerOnlyWhenMoving := FALSE;
	GVL.g_aVisionTrackingSourceConfigA[1].MinimumTriggerVelocityMMs := 1.0;



    //=========================================================================
    // CAMERA 2
    //=========================================================================
    //GVL.g_aVisionConfig[2].Enable := FALSE;
    GVL.g_aVisionConfig[2].CameraID := 2;
    GVL.g_aVisionConfig[2].BaseAddress := 300;
    GVL.g_aVisionConfig[2].CommandOffset := 0;
    GVL.g_aVisionConfig[2].StatusOffset := 100;
    GVL.g_aVisionConfig[2].HeaderOffset := 101;
    GVL.g_aVisionConfig[2].DataOffset := 116;
    //GVL.g_aVisionConfig[2].PositionScale := 0.001;
    //GVL.g_aVisionConfig[2].AngleScale := 0.001;
    GVL.g_aVisionConfig[2].ScoreScale := 1.0;


    //=========================================================================
    // CAMERA 3
    //=========================================================================
    //GVL.g_aVisionConfig[3].Enable := FALSE;
    GVL.g_aVisionConfig[3].CameraID := 3;
    GVL.g_aVisionConfig[3].BaseAddress := 600;
    GVL.g_aVisionConfig[3].CommandOffset := 0;
    GVL.g_aVisionConfig[3].StatusOffset := 100;
    GVL.g_aVisionConfig[3].HeaderOffset := 101;
    GVL.g_aVisionConfig[3].DataOffset := 116;
    //GVL.g_aVisionConfig[3].PositionScale := 0.001;
    //GVL.g_aVisionConfig[3].AngleScale := 0.001;
    GVL.g_aVisionConfig[3].ScoreScale := 1.0;


    //=========================================================================
    // CAMERA 4
    //=========================================================================
    //GVL.g_aVisionConfig[4].Enable := FALSE;
    GVL.g_aVisionConfig[4].CameraID := 4;
    GVL.g_aVisionConfig[4].BaseAddress := 900;
    GVL.g_aVisionConfig[4].CommandOffset := 0;
    GVL.g_aVisionConfig[4].StatusOffset := 100;
    GVL.g_aVisionConfig[4].HeaderOffset := 101;
    GVL.g_aVisionConfig[4].DataOffset := 116;
    //GVL.g_aVisionConfig[4].PositionScale := 0.001;
    //GVL.g_aVisionConfig[4].AngleScale := 0.001;
    GVL.g_aVisionConfig[4].ScoreScale := 1.0;
	
	//=========================================================================
	// CAMERA 1
	//=========================================================================
	//GVL.g_aVisionConfig[1].Robot := E_VisionRobot.VIS_ROBOT_A;
	
	//=========================================================================
	// CAMERA 2
	//=========================================================================
	//GVL.g_aVisionConfig[2].Robot := E_VisionRobot.VIS_ROBOT_A;
	
	//=========================================================================
	// CAMERA 3
	//=========================================================================
	//GVL.g_aVisionConfig[3].Robot := E_VisionRobot.VIS_ROBOT_A;
	
	//=========================================================================
	// CAMERA 4
	//=========================================================================
	//GVL.g_aVisionConfig[4].Robot := E_VisionRobot.VIS_ROBOT_NONE;


    // Đánh dấu đã khởi tạo để không ghi lại mỗi scan.
    xInitialized := TRUE;

END_IF;

END_PROGRAM

// Just_Motion_Control_x86_64_Linux_SM_WV/Application/PRG_MACHINE/POU_CAM
PROGRAM POU_CAM
VAR
	RB_A_READ_CAM, RB_B_READ_CAM   	 : FB_Real_TO_Word_;
	RB_T1_WRITE, RB_T2_WRITE , RB_T1_READ_CAM_OFFSET , RB_T2_READ_CAM_OFFSET			 : FB_word_TO_real_;
	Connect_fail, bit_TRANS_modbus1, bit_RECEI_modbus1 : BOOL;
	TRIGGER_TOP, TRIGGER_DONE, Trigger_Busy : BOOL;
	R_Trig_TriggerDone : R_TRIG;
	T1,T2,T3,T4 : TON;
	i_Vs : INT;
	

END_VAR
VAR // added by the converter: edge detectors and wires of the graphical bodies
    _w1, _w2 : BOOL;
END_VAR

// // check Connect	
// bit_RECEI_modbus1 := GVL.MODBUS[100].0 OR GVL.MODBUS[100 + GVL.NB_Register_Modbus_VS *1].0 OR GVL.MODBUS[100 + GVL.NB_Register_Modbus_VS *2].0 OR GVL.MODBUS[100 + GVL.NB_Register_Modbus_VS *3].0;
// GVL.MODBUS[0].0 := bit_TRANS_modbus1;
// GVL.MODBUS[GVL.NB_Register_Modbus_VS *1].0 := bit_TRANS_modbus1;
// GVL.MODBUS[GVL.NB_Register_Modbus_VS *2].0 := bit_TRANS_modbus1;
// GVL.MODBUS[GVL.NB_Register_Modbus_VS *3].0 := bit_TRANS_modbus1;
// 
// /// Bit control Robot - VS
// i_Vs := 0;
// FOR i_Vs := 0 TO 2 BY 1 DO
// 	IF GVL.Data_Calib_RB[i_Vs].Use THEN
// 		// Tin hieu Trigger Modbus
// 		GVL.MODBUS[GVL.NB_Register_Modbus_VS *i_Vs].1 := GVL.Man_Calib_RB[i_Vs].Trigger_VS OR GVL.Auto_VS_RB[i_Vs].Trigger_VS;
// 		// Tin hieu bao Chay xong cac vi tri calib
// 		GVL.MODBUS[GVL.NB_Register_Modbus_VS *i_Vs].2 := GVL.Man_Calib_RB[i_Vs].Run_Pos_Calib_Done OR GVL.Auto_VS_RB[i_Vs].Run_Pos_Calib_Done;
// 		// Tin hieu bao Trigger Done tu VS System
// 		GVL.Man_Calib_RB[i_Vs].Trigger_Done := GVL.MODBUS[GVL.NB_Register_Modbus_VS *i_Vs + 100].1;
// 		GVL.Auto_VS_RB[i_Vs].Trigger_Done := GVL.MODBUS[GVL.NB_Register_Modbus_VS *i_Vs + 100].1;
// 		// Tin hieu bao Calib Done tu VS System
// 		GVL.Man_Calib_RB[i_Vs].Calib_VS_Done := GVL.MODBUS[GVL.NB_Register_Modbus_VS *i_Vs + 100].2;
// 		GVL.Auto_VS_RB[i_Vs].Calib_VS_Done := GVL.MODBUS[GVL.NB_Register_Modbus_VS *i_Vs + 100].2;		
// 	END_IF
// END_FOR
// // GVL.MODBUS[0].1 := TRIGGER_TOP;
// IF (GVL.MODBUS[0].1) THEN
// 	Trigger_Busy := TRUE;
// ELSE
// 	Trigger_Busy := FALSE;
// END_IF;
// //TRIGGER_DONE := GVL.MODBUS[100].1; // doc tin hieu bao trigger done
// // R_Trig_TriggerDone(CLK := GVL.MODBUS[100].1 );
// // IF Trigger_Busy AND R_Trig_TriggerDone.Q AND NOT GVL.X[8]  THEN
// // 	TRIGGER_DONE := TRUE;
// // END_IF
// 
// //TRIGGER_DONE := GVL.MODBUS[100].1;
// 
// GVL.Pro4_.Auto.Result_Trigger_Vs_Align_Done := TRIGGER_DONE;
// GVL.Pro4_.Man.Result_Trigger_Vs_Align_Done := TRIGGER_DONE;
// //  Bit control - Calib
// //GVL.MODBUS[0].2 := GVL.Pro4_.Man.Run_Calib_Pos_Done;
// GVL.Pro4_.Man.Result_Calib_Done := GVL.MODBUS[100].2;
// 
// 
// 
// // Funtion run
// ACT_TRIGGER_TOP();
// ACT_CHECKCONNECT();
// //ACT_Total();
// 
// 
// // 	RB_A_READ_CAM(	R_RB_X	:= TO_REAL(GVL.RB_A_.CUR_X),
// // 					R_RB_Y	:= TO_REAL(GVL.RB_A_.CUR_Y),
// // 					R_RB_r	:= TO_REAL(GVL.RB_A_.CUR_R),
// // 					LOW_RB_X	=> GVL.MODBUS[2],
// // 					HIGH_RB_X	=> GVL.MODBUS[3],
// // 					LOW_RB_Y	=> GVL.MODBUS[4],
// // 					HIGH_RB_Y	=> GVL.MODBUS[5],
// // 					LOW_RB_R	=> GVL.MODBUS[6],
// // 					HIGH_RB_R	=> GVL.MODBUS[7]);								
// // 	RB_B_READ_CAM(	R_RB_X	:= TO_REAL(GVL.RB_B_.CUR_X),
// // 					R_RB_Y	:= TO_REAL(GVL.RB_B_.CUR_Y),
// // 					R_RB_r	:= TO_REAL(GVL.RB_B_.CUR_R),
// // 					LOW_RB_X	=> GVL.MODBUS[8],
// // 					HIGH_RB_X	=> GVL.MODBUS[9],
// // 					LOW_RB_Y	=> GVL.MODBUS[10],
// // 					HIGH_RB_Y	=> GVL.MODBUS[11],
// // 					LOW_RB_R	=> GVL.MODBUS[12],
// // 					HIGH_RB_R	=> GVL.MODBUS[13]);	
// 								
// RB_T1_WRITE(W_LOW_CAM_X := GVL.MODBUS[102],
// 			W_HIGH_CAM_X := GVL.MODBUS[103],
// 			W_LOW_CAM_Y := GVL.MODBUS[104],
// 			W_HIGH_CAM_Y := GVL.MODBUS[105],
// 			W_LOW_CAM_R := GVL.MODBUS[106],
// 			W_HIGH_CAM_R := GVL.MODBUS[107],
// 			CAM_X	=> GVL.Cam_T1.POS_X_OFFSET,
// 			CAM_Y	=> GVL.Cam_T1.POS_Y_OFFSET,
// 			CAM_R	=> GVL.Cam_T1.POS_R_OFFSET);
// 
// IF (TRIGGER_DONE) THEN
// 	GVL.Pro4_.Auto.Result_Trigger_Vs_Align_Done := TRUE;
// 	GVL.Pro4_.Man.Result_Trigger_Vs_Align_Done := TRUE;
// END_IF;		
// // 	RB_T1_READ_CAM_OFFSET(	W_LOW_CAM_X := GVL.MODBUS[114],
// // 							W_HIGH_CAM_X := GVL.MODBUS[115],
// // 							W_LOW_CAM_Y := GVL.MODBUS[116],
// // 							W_HIGH_CAM_Y := GVL.MODBUS[117],
// // 							W_LOW_CAM_R := GVL.MODBUS[118],
// // 							W_HIGH_CAM_R := GVL.MODBUS[119],
// // 							CAM_X	=> GVL.Cam_T1.POS_X_OFFSET,
// // 							CAM_Y	=> GVL.Cam_T1.POS_Y_OFFSET,
// // 							CAM_R	=> GVL.Cam_T1.POS_R_OFFSET);	
// 			
// // 	RB_T2_WRITE(	W_LOW_CAM_X := GVL.MODBUS[108],
// // 				W_HIGH_CAM_X := GVL.MODBUS[109],
// // 				W_LOW_CAM_Y := GVL.MODBUS[110],
// // 				W_HIGH_CAM_Y := GVL.MODBUS[111],
// // 				W_LOW_CAM_R := GVL.MODBUS[112],
// // 				W_HIGH_CAM_R := GVL.MODBUS[113],
// // 				CAM_X	=> GVL.Cam_T2.Pos_X,
// // 				CAM_Y	=> GVL.Cam_T2.Pos_Y,
// // 				CAM_R	=> GVL.Cam_T2.Pos_R);
// 				
// // 	RB_T2_READ_CAM_OFFSET(	W_LOW_CAM_X := GVL.MODBUS[120],
// // 							W_HIGH_CAM_X := GVL.MODBUS[121],
// // 							W_LOW_CAM_Y := GVL.MODBUS[122],
// // 							W_HIGH_CAM_Y := GVL.MODBUS[123],
// // 							W_LOW_CAM_R := GVL.MODBUS[124],
// // 							W_HIGH_CAM_R := GVL.MODBUS[125],
// // 							CAM_X	=> GVL.Cam_T2.POS_X_OFFSET,
// // 							CAM_Y	=> GVL.Cam_T2.POS_Y_OFFSET,
// // 							CAM_R	=> GVL.Cam_T2.POS_R_OFFSET);

ACTION ACT_CHECKCONNECT:
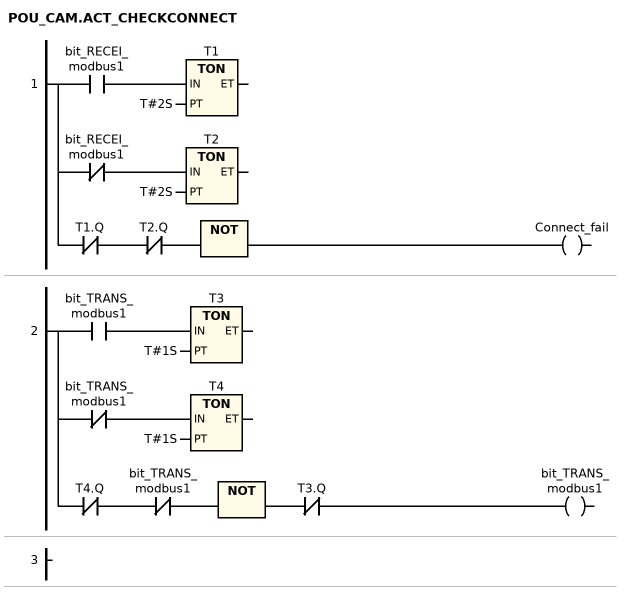
// NETWORK 1
T1(IN := bit_RECEI_modbus1, PT := T#2S); // TON
T2(IN := NOT bit_RECEI_modbus1, PT := T#2S); // TON
Connect_fail := NOT (NOT T1.Q AND NOT T2.Q);

// NETWORK 2
T3(IN := bit_TRANS_modbus1, PT := T#1S); // TON
T4(IN := NOT bit_TRANS_modbus1, PT := T#1S); // TON
bit_TRANS_modbus1 := NOT (NOT T4.Q AND NOT bit_TRANS_modbus1) AND NOT T3.Q;

// NETWORK 3
END_ACTION

ACTION ACT_Total:
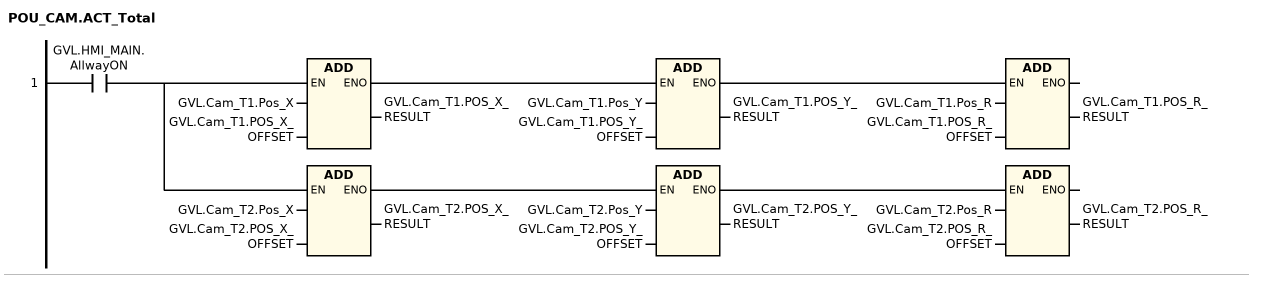
// NETWORK 1
_w1 := GVL.HMI_MAIN.AllwayON;
IF _w1 THEN GVL.Cam_T1.POS_X_RESULT := GVL.Cam_T1.Pos_X + GVL.Cam_T1.POS_X_OFFSET; END_IF
IF _w1 THEN GVL.Cam_T1.POS_Y_RESULT := GVL.Cam_T1.Pos_Y + GVL.Cam_T1.POS_Y_OFFSET; END_IF
IF _w1 THEN GVL.Cam_T1.POS_R_RESULT := GVL.Cam_T1.Pos_R + GVL.Cam_T1.POS_R_OFFSET; END_IF
_w2 := GVL.HMI_MAIN.AllwayON;
IF _w2 THEN GVL.Cam_T2.POS_X_RESULT := GVL.Cam_T2.Pos_X + GVL.Cam_T2.POS_X_OFFSET; END_IF
IF _w2 THEN GVL.Cam_T2.POS_Y_RESULT := GVL.Cam_T2.Pos_Y + GVL.Cam_T2.POS_Y_OFFSET; END_IF
IF _w2 THEN GVL.Cam_T2.POS_R_RESULT := GVL.Cam_T2.Pos_R + GVL.Cam_T2.POS_R_OFFSET; END_IF
END_ACTION

ACTION ACT_TRIGGER_TOP:
TRIGGER_TOP := (GVL.MB_[10] AND GVL.RB_B.Manual) OR
				 (GVL.Pro4_.Auto.Trigger_Vs_Align_On_Off) OR GVL.Pro4_.Man.Trigger_Vs_Align_On_Off; // trigger auto VS align

GVL.MB_[50] := GVL.MODBUS[100].5 ;
GVL.MB_[51] := GVL.MODBUS[100].6 ;
GVL.MB_[52] := GVL.MODBUS[100].7 ;
GVL.MB_[53] := GVL.MODBUS[100].8 ;

GVL.MB_[54] := GVL.MODBUS[100].12 ;
GVL.MB_[55] := GVL.MODBUS[100].13 ;
GVL.MB_[56] := GVL.MODBUS[100].14 ;
GVL.MB_[57] := GVL.MODBUS[100].15 ;
END_ACTION

END_PROGRAM

// Just_Motion_Control_x86_64_Linux_SM_WV/Application/FB_/FB_word_TO_real_
FUNCTION_BLOCK FB_word_TO_real_
VAR_INPUT
	W_LOW_CAM_X, W_HIGH_CAM_X,
	W_LOW_CAM_Y, W_HIGH_CAM_Y,
	W_LOW_CAM_R, W_HIGH_CAM_R : WORD;
END_VAR
VAR_OUTPUT
	CAM_X, CAM_Y, CAM_R : REAL;
END_VAR
VAR
	DINT_cam_X, DINT_cam_Y, DINT_cam_R : DINT;
END_VAR

	DINT_cam_X := DWORD_TO_DINT(SHL(WORD_TO_DWORD(W_HIGH_CAM_X),16) OR WORD_TO_DWORD(W_LOW_CAM_X));
	DINT_cam_Y := DWORD_TO_DINT(SHL(WORD_TO_DWORD(W_HIGH_CAM_Y),16) OR WORD_TO_DWORD(W_LOW_CAM_Y));
	DINT_cam_R := DWORD_TO_DINT(SHL(WORD_TO_DWORD(W_HIGH_CAM_R),16) OR WORD_TO_DWORD(W_LOW_CAM_R));
	
	CAM_X := DINT_TO_REAL(DINT_cam_X)/1000;

	CAM_Y := DINT_TO_REAL(DINT_cam_Y)/1000;

	CAM_R := DINT_TO_REAL(DINT_cam_R)/1000;

END_FUNCTION_BLOCK

// Just_Motion_Control_x86_64_Linux_SM_WV/Application/PRG_MACHINE/PRG_VisionModbus
PROGRAM PRG_VisionModbus
VAR
	fbVisionModbus : ARRAY[1..GVL.C_MAX_VISION_CHANNELS] OF FB_VisionModbusDriver;
	uiCamera : UINT;
	xManualTriggerActive : ARRAY[1..GVL.C_MAX_VISION_CHANNELS] OF BOOL; // Manual HMI đang sở hữu Trigger của Camera.
END_VAR

//=============================================================================
// PRG_VisionModbus
//----------------------------------------------------------------------------- 
// Thêm PRG này vào Task_Communication, sau POU_MODBUS.
//=============================================================================
FOR uiCamera := 1 TO GVL.C_MAX_VISION_CHANNELS DO
	//=============================================================================
	// MANUAL TRIGGER HMI
	//-----------------------------------------------------------------------------
	// ON  : Manual chiếm quyền và giữ Execute TRUE.
	// OFF : Nếu trước đó Manual đang chiếm quyền thì hạ Execute FALSE và trả quyền.
	// Auto không bị ảnh hưởng khi Manual chưa từng chiếm quyền.
	//=============================================================================
	IF GVL.Man_Calib_RB[uiCamera].Trigger_VS THEN
	
		// HMI đang ON -> Manual sở hữu Trigger.
		xManualTriggerActive[uiCamera] := TRUE;
	
		// Giữ Trigger ON liên tục.
		GVL.g_aVisionCommand[uiCamera].Execute := TRUE;
	
	ELSIF xManualTriggerActive[uiCamera] THEN
	
		// HMI vừa chuyển OFF -> hạ Trigger.
		GVL.g_aVisionCommand[uiCamera].Execute := FALSE;
	
		// Trả quyền điều khiển cho Auto.
		xManualTriggerActive[uiCamera] := FALSE;
	
	END_IF;

    fbVisionModbus[uiCamera](
        Enable := GVL.g_aVisionConfig[uiCamera].Enable,
        Reset := GVL.g_aVisionCommand[uiCamera].Reset,
        Config := GVL.g_aVisionConfig[uiCamera],
        Command := GVL.g_aVisionCommand[uiCamera],
        ModbusControl := GVL.g_aVisionModbusControl[uiCamera],
        ChannelStatus := GVL.g_aVisionStatus[uiCamera],
        ModbusStatus := GVL.g_aVisionModbusStatus[uiCamera],
        VisionResult := GVL.g_aVisionResult[uiCamera],
        Registers := GVL.MODBUS
    );
END_FOR;

END_PROGRAM

// Just_Motion_Control_x86_64_Linux_SM_WV/Application/PRG_ROBOT/PRG_VisionManager
PROGRAM PRG_VisionManager
VAR
    //=========================================================================
    // VISION ALIGN FUNCTION BLOCKS
    //-------------------------------------------------------------------------
    // Mỗi Camera có một instance FB_VisionAlign riêng.
    // Vì FB có State/Timer/TriggerID nội bộ nên tuyệt đối không dùng chung
    // một instance cho nhiều Camera.
    //=========================================================================
    fbVisionAlign : ARRAY[1..GVL.C_MAX_VISION_CHANNELS] OF FB_VisionAlign;

    //=========================================================================
    // CAMERA RUNTIME
    // Mỗi phần tử Array tương ứng với một Camera.
    //=========================================================================
    xStartAlign : ARRAY[1..GVL.C_MAX_VISION_CHANNELS] OF BOOL;             // Start của FB_VisionAlign từng Camera.
    uiJobID : ARRAY[1..GVL.C_MAX_VISION_CHANNELS] OF UINT;                 // JobID đã latch khi nhận Request.
    eRequester : ARRAY[1..GVL.C_MAX_VISION_CHANNELS] OF E_VisionRobot;     // Robot đang sở hữu Camera.
    iState : ARRAY[1..GVL.C_MAX_VISION_CHANNELS] OF INT;                   // State transaction riêng từng Camera.

    //=========================================================================
    // LOOP VARIABLE
    //=========================================================================
    uiCamera : UINT;                                                        // Camera index dùng trong vòng FOR.
	wControl_Tmp : WORD;
    wStatus_Tmp : WORD;
END_VAR

//=============================================================================
// PRG_VisionManager
//=============================================================================
// Chức năng:
// - Nhận Vision Align Request từ Robot A và Robot B.
// - Kiểm tra CameraID, Enable và Robot Assignment.
// - Mỗi Camera chỉ có một Robot sở hữu tại một thời điểm.
// - Điều khiển FB_VisionAlign riêng của từng Camera.
// - Trả Done / Error / Result về đúng Robot đã gửi Request.
//
// STATE:
// 0   = IDLE
// 10  = START VISION ALIGN
// 20  = WAIT VISION RESULT
// 30  = DONE - WAIT ROBOT RELEASE
// 900 = ERROR - WAIT ROBOT RELEASE
//=============================================================================


//=============================================================================
// 1. RESET REQUEST A SAU KHI ROBOT ĐÃ HẠ EXECUTE
//-----------------------------------------------------------------------------
// Phần này chủ yếu xử lý các lỗi xảy ra trước khi Camera được chiếm quyền,
// ví dụ CameraID sai, Camera Disable hoặc Camera không thuộc Robot A.
//=============================================================================
IF NOT GVL.g_stVisionAlignRequestA.Execute
AND NOT GVL.g_stVisionAlignRequestA.Busy
AND GVL.g_stVisionAlignRequestA.Error THEN
    GVL.g_stVisionAlignRequestA.Error := FALSE;
    GVL.g_stVisionAlignRequestA.ErrorID := 0;
    GVL.g_stVisionAlignRequestA.Done := FALSE;
    GVL.g_stVisionAlignRequestA.ResultOK := FALSE;
    GVL.g_stVisionAlignRequestA.ResultValid := FALSE;
END_IF;


//=============================================================================
// 2. RESET REQUEST B SAU KHI ROBOT ĐÃ HẠ EXECUTE
//=============================================================================
IF NOT GVL.g_stVisionAlignRequestB.Execute
AND NOT GVL.g_stVisionAlignRequestB.Busy
AND GVL.g_stVisionAlignRequestB.Error THEN
    GVL.g_stVisionAlignRequestB.Error := FALSE;
    GVL.g_stVisionAlignRequestB.ErrorID := 0;
    GVL.g_stVisionAlignRequestB.Done := FALSE;
    GVL.g_stVisionAlignRequestB.ResultOK := FALSE;
    GVL.g_stVisionAlignRequestB.ResultValid := FALSE;
END_IF;


//=============================================================================
// 3. NHẬN REQUEST TỪ ROBOT A
//=============================================================================
IF GVL.g_stVisionAlignRequestA.Execute
AND NOT GVL.g_stVisionAlignRequestA.Busy
AND NOT GVL.g_stVisionAlignRequestA.Done
AND NOT GVL.g_stVisionAlignRequestA.Error THEN

    //-------------------------------------------------------------------------
    // Kiểm tra CameraID trước khi dùng CameraID làm Array Index.
    //-------------------------------------------------------------------------
    IF (GVL.g_stVisionAlignRequestA.CameraID < 1)
    OR (GVL.g_stVisionAlignRequestA.CameraID > GVL.C_MAX_VISION_CHANNELS) THEN
        GVL.g_stVisionAlignRequestA.Error := TRUE;
        GVL.g_stVisionAlignRequestA.ErrorID := 1;

    ELSE
        uiCamera := GVL.g_stVisionAlignRequestA.CameraID;

        //-------------------------------------------------------------------------
        // Camera phải được Enable.
        //-------------------------------------------------------------------------
        IF NOT GVL.g_aVisionConfig[uiCamera].Enable THEN
            GVL.g_stVisionAlignRequestA.Error := TRUE;
            GVL.g_stVisionAlignRequestA.ErrorID := 2;

        //-------------------------------------------------------------------------
        // Camera phải được cấu hình thuộc Robot A.
        //-------------------------------------------------------------------------
        ELSIF GVL.g_aVisionConfig[uiCamera].Robot <> E_VisionRobot.VIS_ROBOT_A THEN
            GVL.g_stVisionAlignRequestA.Error := TRUE;
            GVL.g_stVisionAlignRequestA.ErrorID := 3;

        //-------------------------------------------------------------------------
        // Camera phải đang rảnh.
        //-------------------------------------------------------------------------
        ELSIF eRequester[uiCamera] <> E_VisionRobot.VIS_ROBOT_NONE THEN
            GVL.g_stVisionAlignRequestA.Error := TRUE;
            GVL.g_stVisionAlignRequestA.ErrorID := 4;

        ELSE
            // Latch JobID để dữ liệu Request thay đổi bên ngoài không ảnh hưởng
            // transaction đang chạy.
            uiJobID[uiCamera] := GVL.g_stVisionAlignRequestA.JobID;

            // Robot A chiếm quyền Camera.
            eRequester[uiCamera] := E_VisionRobot.VIS_ROBOT_A;

            // Xóa status/result cũ trước transaction mới.
            GVL.g_stVisionAlignRequestA.Busy := TRUE;
            GVL.g_stVisionAlignRequestA.Done := FALSE;
            GVL.g_stVisionAlignRequestA.Error := FALSE;
            GVL.g_stVisionAlignRequestA.ErrorID := 0;
            GVL.g_stVisionAlignRequestA.ResultOK := FALSE;
            GVL.g_stVisionAlignRequestA.ResultValid := FALSE;
            GVL.g_stVisionAlignRequestA.TriggerID := 0;
            GVL.g_stVisionAlignRequestA.X := 0.0;
            GVL.g_stVisionAlignRequestA.Y := 0.0;
            GVL.g_stVisionAlignRequestA.Z := 0.0;
            GVL.g_stVisionAlignRequestA.A := 0.0;
            GVL.g_stVisionAlignRequestA.Score := 0.0;
            GVL.g_stVisionAlignRequestA.FeatureID := 0;

            // Bắt đầu transaction của Camera này.
            iState[uiCamera] := 10;
        END_IF;
    END_IF;
END_IF;


//=============================================================================
// 4. NHẬN REQUEST TỪ ROBOT B
//=============================================================================
IF GVL.g_stVisionAlignRequestB.Execute
AND NOT GVL.g_stVisionAlignRequestB.Busy
AND NOT GVL.g_stVisionAlignRequestB.Done
AND NOT GVL.g_stVisionAlignRequestB.Error THEN

    //-------------------------------------------------------------------------
    // Kiểm tra CameraID trước khi dùng làm Array Index.
    //-------------------------------------------------------------------------
    IF (GVL.g_stVisionAlignRequestB.CameraID < 1)
    OR (GVL.g_stVisionAlignRequestB.CameraID > GVL.C_MAX_VISION_CHANNELS) THEN
        GVL.g_stVisionAlignRequestB.Error := TRUE;
        GVL.g_stVisionAlignRequestB.ErrorID := 1;

    ELSE
        uiCamera := GVL.g_stVisionAlignRequestB.CameraID;

        //-------------------------------------------------------------------------
        // Camera phải được Enable.
        //-------------------------------------------------------------------------
        IF NOT GVL.g_aVisionConfig[uiCamera].Enable THEN
            GVL.g_stVisionAlignRequestB.Error := TRUE;
            GVL.g_stVisionAlignRequestB.ErrorID := 2;

        //-------------------------------------------------------------------------
        // Camera phải được cấu hình thuộc Robot B.
        //-------------------------------------------------------------------------
        ELSIF GVL.g_aVisionConfig[uiCamera].Robot <> E_VisionRobot.VIS_ROBOT_B THEN
            GVL.g_stVisionAlignRequestB.Error := TRUE;
            GVL.g_stVisionAlignRequestB.ErrorID := 3;

        //-------------------------------------------------------------------------
        // Camera phải đang rảnh.
        //-------------------------------------------------------------------------
        ELSIF eRequester[uiCamera] <> E_VisionRobot.VIS_ROBOT_NONE THEN
            GVL.g_stVisionAlignRequestB.Error := TRUE;
            GVL.g_stVisionAlignRequestB.ErrorID := 4;

        ELSE
            // Latch JobID.
            uiJobID[uiCamera] := GVL.g_stVisionAlignRequestB.JobID;

            // Robot B chiếm quyền Camera.
            eRequester[uiCamera] := E_VisionRobot.VIS_ROBOT_B;

            // Xóa status/result cũ.
            GVL.g_stVisionAlignRequestB.Busy := TRUE;
            GVL.g_stVisionAlignRequestB.Done := FALSE;
            GVL.g_stVisionAlignRequestB.Error := FALSE;
            GVL.g_stVisionAlignRequestB.ErrorID := 0;
            GVL.g_stVisionAlignRequestB.ResultOK := FALSE;
            GVL.g_stVisionAlignRequestB.ResultValid := FALSE;
            GVL.g_stVisionAlignRequestB.TriggerID := 0;
            GVL.g_stVisionAlignRequestB.X := 0.0;
            GVL.g_stVisionAlignRequestB.Y := 0.0;
            GVL.g_stVisionAlignRequestB.Z := 0.0;
            GVL.g_stVisionAlignRequestB.A := 0.0;
            GVL.g_stVisionAlignRequestB.Score := 0.0;
            GVL.g_stVisionAlignRequestB.FeatureID := 0;

            // Bắt đầu transaction.
            iState[uiCamera] := 10;
        END_IF;
    END_IF;
END_IF;


//=============================================================================
// 5. XỬ LÝ STATE CỦA TỪNG CAMERA
//=============================================================================
FOR uiCamera := 1 TO GVL.C_MAX_VISION_CHANNELS DO

    CASE iState[uiCamera] OF

        //=====================================================================
        // STATE 0 - IDLE
        //=====================================================================
        0:
            xStartAlign[uiCamera] := FALSE;

        //=====================================================================
        // STATE 10 - START VISION ALIGN
        //-------------------------------------------------------------------------
        // Start được giữ TRUE trong suốt transaction.
        // FB_VisionAlign tự xử lý Trigger -> Wait Result -> Done/Error.
        //=====================================================================
        10:
            xStartAlign[uiCamera] := TRUE;
            iState[uiCamera] := 20;

        //=====================================================================
        // STATE 20 - WAIT RESULT
        //-------------------------------------------------------------------------
        // Không xử lý output tại đây.
        // FB được gọi ở phần 6.
        // Output FB được đọc ở phần 7 sau khi FB đã được scan.
        //=====================================================================
        20:
            ;

        //=====================================================================
        // STATE 30 - DONE / WAIT ROBOT RELEASE
        //=====================================================================
        30:
            xStartAlign[uiCamera] := FALSE;

            CASE eRequester[uiCamera] OF

                // Robot A đã nhận Done và hạ Execute.
                E_VisionRobot.VIS_ROBOT_A:
                    IF NOT GVL.g_stVisionAlignRequestA.Execute THEN
                        GVL.g_stVisionAlignRequestA.Busy := FALSE;
                        GVL.g_stVisionAlignRequestA.Done := FALSE;
                        GVL.g_stVisionAlignRequestA.Error := FALSE;
                        GVL.g_stVisionAlignRequestA.ErrorID := 0;

                        eRequester[uiCamera] := E_VisionRobot.VIS_ROBOT_NONE;
                        uiJobID[uiCamera] := 0;
                        iState[uiCamera] := 0;
                    END_IF;

                // Robot B đã nhận Done và hạ Execute.
                E_VisionRobot.VIS_ROBOT_B:
                    IF NOT GVL.g_stVisionAlignRequestB.Execute THEN
                        GVL.g_stVisionAlignRequestB.Busy := FALSE;
                        GVL.g_stVisionAlignRequestB.Done := FALSE;
                        GVL.g_stVisionAlignRequestB.Error := FALSE;
                        GVL.g_stVisionAlignRequestB.ErrorID := 0;

                        eRequester[uiCamera] := E_VisionRobot.VIS_ROBOT_NONE;
                        uiJobID[uiCamera] := 0;
                        iState[uiCamera] := 0;
                    END_IF;

                ELSE
                    // Safety fallback: Camera không có owner hợp lệ.
                    xStartAlign[uiCamera] := FALSE;
                    eRequester[uiCamera] := E_VisionRobot.VIS_ROBOT_NONE;
                    uiJobID[uiCamera] := 0;
                    iState[uiCamera] := 0;
            END_CASE;

        //=====================================================================
        // STATE 900 - ERROR / WAIT ROBOT RELEASE
        //=====================================================================
        900:
            xStartAlign[uiCamera] := FALSE;

            CASE eRequester[uiCamera] OF

                // Robot A xác nhận Error bằng cách hạ Execute.
                E_VisionRobot.VIS_ROBOT_A:
                    IF NOT GVL.g_stVisionAlignRequestA.Execute THEN
                        GVL.g_stVisionAlignRequestA.Busy := FALSE;
                        GVL.g_stVisionAlignRequestA.Done := FALSE;
                        GVL.g_stVisionAlignRequestA.Error := FALSE;
                        GVL.g_stVisionAlignRequestA.ErrorID := 0;

                        eRequester[uiCamera] := E_VisionRobot.VIS_ROBOT_NONE;
                        uiJobID[uiCamera] := 0;
                        iState[uiCamera] := 0;
                    END_IF;

                // Robot B xác nhận Error bằng cách hạ Execute.
                E_VisionRobot.VIS_ROBOT_B:
                    IF NOT GVL.g_stVisionAlignRequestB.Execute THEN
                        GVL.g_stVisionAlignRequestB.Busy := FALSE;
                        GVL.g_stVisionAlignRequestB.Done := FALSE;
                        GVL.g_stVisionAlignRequestB.Error := FALSE;
                        GVL.g_stVisionAlignRequestB.ErrorID := 0;

                        eRequester[uiCamera] := E_VisionRobot.VIS_ROBOT_NONE;
                        uiJobID[uiCamera] := 0;
                        iState[uiCamera] := 0;
                    END_IF;

                ELSE
                    // Safety fallback.
                    xStartAlign[uiCamera] := FALSE;
                    eRequester[uiCamera] := E_VisionRobot.VIS_ROBOT_NONE;
                    uiJobID[uiCamera] := 0;
                    iState[uiCamera] := 0;
            END_CASE;

        //=====================================================================
        // INVALID STATE
        //=====================================================================
        ELSE
            xStartAlign[uiCamera] := FALSE;
            eRequester[uiCamera] := E_VisionRobot.VIS_ROBOT_NONE;
            uiJobID[uiCamera] := 0;
            iState[uiCamera] := 0;

    END_CASE;

END_FOR;


//=============================================================================
// 6. GỌI FB_VISIONALIGN CHO TẤT CẢ CAMERA
//-----------------------------------------------------------------------------
// BẮT BUỘC gọi mỗi instance ở mọi PLC scan.
//=============================================================================
FOR uiCamera := 1 TO GVL.C_MAX_VISION_CHANNELS DO

    fbVisionAlign[uiCamera](
        Enable := GVL.g_aVisionConfig[uiCamera].Enable,
        Start := xStartAlign[uiCamera],
        CameraID := uiCamera,
        JobID := uiJobID[uiCamera]
    );

END_FOR;


//=============================================================================
// 7. ĐỌC OUTPUT FB SAU KHI FB ĐÃ ĐƯỢC SCAN
//=============================================================================
FOR uiCamera := 1 TO GVL.C_MAX_VISION_CHANNELS DO

    IF iState[uiCamera] = 20 THEN

        //=====================================================================
        // TRANSACTION DONE
        //=====================================================================
        IF fbVisionAlign[uiCamera].Done THEN

            CASE eRequester[uiCamera] OF

                //-------------------------------------------------------------
                // RESULT -> ROBOT A
                //-------------------------------------------------------------
                E_VisionRobot.VIS_ROBOT_A:
                    GVL.g_stVisionAlignRequestA.TriggerID := fbVisionAlign[uiCamera].TriggerID;
                    GVL.g_stVisionAlignRequestA.X := fbVisionAlign[uiCamera].VisionX;
                    GVL.g_stVisionAlignRequestA.Y := fbVisionAlign[uiCamera].VisionY;
                    GVL.g_stVisionAlignRequestA.Z := fbVisionAlign[uiCamera].VisionZ;
                    GVL.g_stVisionAlignRequestA.A := fbVisionAlign[uiCamera].VisionA;
                    GVL.g_stVisionAlignRequestA.Score := fbVisionAlign[uiCamera].VisionScore;
                    GVL.g_stVisionAlignRequestA.FeatureID := fbVisionAlign[uiCamera].VisionFeatureID;
                    GVL.g_stVisionAlignRequestA.ResultValid := fbVisionAlign[uiCamera].ResultValid;
                    GVL.g_stVisionAlignRequestA.ResultStatus := fbVisionAlign[uiCamera].ResultStatus;

                    // Business result:
                    // OK -> TRUE.
                    // NG/NOT_FOUND/... -> FALSE nhưng transaction vẫn Done.
                    GVL.g_stVisionAlignRequestA.ResultOK :=
                        fbVisionAlign[uiCamera].ResultStatus = E_VisionResultStatus.VIS_RESULT_OK;

                    GVL.g_stVisionAlignRequestA.Busy := FALSE;
                    GVL.g_stVisionAlignRequestA.Error := FALSE;
                    GVL.g_stVisionAlignRequestA.ErrorID := 0;
                    GVL.g_stVisionAlignRequestA.Done := TRUE;

                //-------------------------------------------------------------
                // RESULT -> ROBOT B
                //-------------------------------------------------------------
                E_VisionRobot.VIS_ROBOT_B:
                    GVL.g_stVisionAlignRequestB.TriggerID := fbVisionAlign[uiCamera].TriggerID;
                    GVL.g_stVisionAlignRequestB.X := fbVisionAlign[uiCamera].VisionX;
                    GVL.g_stVisionAlignRequestB.Y := fbVisionAlign[uiCamera].VisionY;
                    GVL.g_stVisionAlignRequestB.Z := fbVisionAlign[uiCamera].VisionZ;
                    GVL.g_stVisionAlignRequestB.A := fbVisionAlign[uiCamera].VisionA;
                    GVL.g_stVisionAlignRequestB.Score := fbVisionAlign[uiCamera].VisionScore;
                    GVL.g_stVisionAlignRequestB.FeatureID := fbVisionAlign[uiCamera].VisionFeatureID;
                    GVL.g_stVisionAlignRequestB.ResultValid := fbVisionAlign[uiCamera].ResultValid;
                    GVL.g_stVisionAlignRequestB.ResultStatus := fbVisionAlign[uiCamera].ResultStatus;

                    GVL.g_stVisionAlignRequestB.ResultOK :=
                        fbVisionAlign[uiCamera].ResultStatus = E_VisionResultStatus.VIS_RESULT_OK;

                    GVL.g_stVisionAlignRequestB.Busy := FALSE;
                    GVL.g_stVisionAlignRequestB.Error := FALSE;
                    GVL.g_stVisionAlignRequestB.ErrorID := 0;
                    GVL.g_stVisionAlignRequestB.Done := TRUE;

            END_CASE;

            // Hạ Start để FB_VisionAlign thoát State Done sau handshake.
            xStartAlign[uiCamera] := FALSE;

            // Giữ Camera cho requester cho tới khi requester hạ Execute.
            iState[uiCamera] := 30;


        //=====================================================================
        // TRANSACTION ERROR
        //=====================================================================
        ELSIF fbVisionAlign[uiCamera].Error THEN

            CASE eRequester[uiCamera] OF

                //-------------------------------------------------------------
                // ERROR -> ROBOT A
                //-------------------------------------------------------------
                E_VisionRobot.VIS_ROBOT_A:
                    GVL.g_stVisionAlignRequestA.Busy := FALSE;
                    GVL.g_stVisionAlignRequestA.Done := FALSE;
                    GVL.g_stVisionAlignRequestA.ResultOK := FALSE;
                    GVL.g_stVisionAlignRequestA.ResultValid := FALSE;
                    GVL.g_stVisionAlignRequestA.Error := TRUE;

                    // 100 + ErrorID để phân biệt lỗi Manager và lỗi FB.
                    GVL.g_stVisionAlignRequestA.ErrorID :=
                        100 + fbVisionAlign[uiCamera].ErrorID;

                //-------------------------------------------------------------
                // ERROR -> ROBOT B
                //-------------------------------------------------------------
                E_VisionRobot.VIS_ROBOT_B:
                    GVL.g_stVisionAlignRequestB.Busy := FALSE;
                    GVL.g_stVisionAlignRequestB.Done := FALSE;
                    GVL.g_stVisionAlignRequestB.ResultOK := FALSE;
                    GVL.g_stVisionAlignRequestB.ResultValid := FALSE;
                    GVL.g_stVisionAlignRequestB.Error := TRUE;

                    GVL.g_stVisionAlignRequestB.ErrorID :=
                        100 + fbVisionAlign[uiCamera].ErrorID;

            END_CASE;

            // Hạ Start để FB bắt đầu reset Error.
            xStartAlign[uiCamera] := FALSE;

            // Camera chỉ được giải phóng sau khi Robot hạ Execute.
            iState[uiCamera] := 900;

        END_IF;

    END_IF;

END_FOR;

// Monitor ControlWord and Status Wword
FOR uiCamera := 1 TO GVL.C_MAX_VISION_CHANNELS DO
	wControl_Tmp := GVL.MODBUS[0 + (uiCamera-1)*300];
 	wStatus_Tmp := GVL.MODBUS[100 + (uiCamera-1)*300];
	GVL.g_aVision_ControlWord[uiCamera].HeartBeat := wControl_Tmp.0;
	GVL.g_aVision_ControlWord[uiCamera].TriggerCam := wControl_Tmp.1;
	GVL.g_aVision_ControlWord[uiCamera].RunCalib := wControl_Tmp.2;
	GVL.g_aVision_ControlWord[uiCamera].CalibPosReady := wControl_Tmp.3;
	GVL.g_aVision_ControlWord[uiCamera].AckResult := wControl_Tmp.4;
	GVL.g_aVision_ControlWord[uiCamera].AckBlock := wControl_Tmp.5;
	GVL.g_aVision_ControlWord[uiCamera].ResetVision := wControl_Tmp.6;
	GVL.g_aVision_ControlWord[uiCamera].AbortVision := wControl_Tmp.7;
	
	GVL.g_aVision_StatusWord[uiCamera].HeartBeat := wStatus_Tmp.0;
	GVL.g_aVision_StatusWord[uiCamera].TriggerDone := wStatus_Tmp.1;
	GVL.g_aVision_StatusWord[uiCamera].CalibDone := wStatus_Tmp.2;
	GVL.g_aVision_StatusWord[uiCamera].ResultReady := wStatus_Tmp.3;
	GVL.g_aVision_StatusWord[uiCamera].Busy := wStatus_Tmp.4;
	GVL.g_aVision_StatusWord[uiCamera].Run1Slot := wStatus_Tmp.5;
	GVL.g_aVision_StatusWord[uiCamera].BlockReady := wStatus_Tmp.6;
	GVL.g_aVision_StatusWord[uiCamera].Error := wStatus_Tmp.7;
	GVL.g_aVision_StatusWord[uiCamera].CalibBusy := wStatus_Tmp.8;
	GVL.g_aVision_StatusWord[uiCamera].CalibError := wStatus_Tmp.9;
	
END_FOR;

END_PROGRAM

// Just_Motion_Control_x86_64_Linux_SM_WV/Application/PRG_MACHINE/POU_Alarm
PROGRAM POU_Alarm
VAR
	T_Alarm : ARRAY [0..100] OF TON;
END_VAR

Alarm_Robot();
IF GVL.ProjectAndModel.Project_No_Current = 3 THEN
	Alarm_Project_4();
END_IF;

ACTION Alarm_Project_4:
// Loi Tin hieu SS Press may TS 1
T_Alarm[50](IN:= ((POU_MOTION.Pro_MC1_4 = 10 AND NOT GVL.Pro4_.Signal_In.T_Ts_Press_Up.Q)) , PT := T#5S); 
IF T_Alarm[50].Q THEN
	GVL.Alarm_P4.Alarm_TS_SS_Up := TRUE;
ELSE
	GVL.Alarm_P4.Alarm_TS_SS_Up := FALSE;
END_IF

// Loi Tin hieu SS Press may VS 1
T_Alarm[51](IN:= ((POU_MOTION.Pro_MC2_4 = 10 AND NOT GVL.Pro4_.Signal_In.T_Vs_detect.Q)) , PT := T#5S); 
IF T_Alarm[51].Q THEN
	GVL.Alarm_P4.Alarm_VS_SS_JigOut := TRUE;
ELSE
	GVL.Alarm_P4.Alarm_VS_SS_JigOut := FALSE;
END_IF

// Loi Tin hieu Pass/Fail Press may TS
T_Alarm[52](IN:= ((POU_MOTION.Pro_MC1_4 = 20 AND POU_MOTION.on_centering = 20 AND GVL.Pro4_.Signal_In.T_Ts_Press_Up.Q AND NOT GVL.Pro4_.Signal_In.T_Ts_Pass.Q AND NOT GVL.Pro4_.Signal_In.T_Ts_Fail.Q)) , PT := T#10S); 
IF T_Alarm[52].Q THEN
	GVL.Alarm_P4.Alarm_TS_NG_Pass_Fail_Signal := TRUE;
ELSE
	GVL.Alarm_P4.Alarm_TS_NG_Pass_Fail_Signal := FALSE;
END_IF

// Loi Tin hieu Pass/Fail Press may VS
T_Alarm[53](IN:= ((POU_MOTION.Pro_MC2_4 = 20 AND POU_MOTION.T_MC2_4.q AND GVL.Pro4_.Signal_In.T_Vs_detect.Q AND NOT GVL.Pro4_.Signal_In.T_Vs_Pass.Q AND NOT GVL.Pro4_.Signal_In.T_Vs_Fail.Q)) , PT := T#10S); 
IF T_Alarm[53].Q THEN
	GVL.Alarm_P4.Alarm_VS_NG_Pass_Fail_Signal := TRUE;
ELSE
	GVL.Alarm_P4.Alarm_VS_NG_Pass_Fail_Signal := FALSE;
END_IF

// Loi qua thoi gian test may Test song
IF POU_MOTION.Pro_MC1_4 = 20 AND POU_MOTION.on_centering = 20 AND NOT GVL.Pro4_.Signal_In.T_Ts_Press_Up.Q AND POU_MOTION.Ton_Limit_Test_TS.Q THEN
	GVL.Alarm_P4.Alarm_Limit_Test_TS := TRUE;
ELSE
	GVL.Alarm_P4.Alarm_Limit_Test_TS := FALSE;
END_IF

// Loi qua thoi gian test may vision
IF POU_MOTION.Pro_MC2_4 = 20 AND POU_MOTION.T_MC2_4.q AND NOT GVL.Pro4_.Signal_In.T_Vs_detect.Q AND POU_MOTION.Ton_Limit_Test_VS.Q THEN
	GVL.Alarm_P4.Alarm_Limit_Test_VS := TRUE;
ELSE
	GVL.Alarm_P4.Alarm_Limit_Test_VS := FALSE;
END_IF

// Loi ko co hang dau vao sau 3P
T_Alarm[54]( IN:= GVL.X[27] AND POU_MOTION.RUN_PROJECT, PT := T#180S);
IF T_Alarm[54].Q THEN
	GVL.Alarm_P4.Wait_Product_Input := TRUE;
ELSE
	GVL.Alarm_P4.Wait_Product_Input := FALSE;
END_IF

// Loi khong do cduoc code may test song
T_Alarm[55]( IN := GVL.Pro4_.Auto.Alarm_Not_barcode, PT := T#1S);
IF T_Alarm[55].Q THEN
	GVL.Alarm_P4.Read_Barcode_TS := TRUE;
ELSE
	GVL.Alarm_P4.Read_Barcode_TS := FALSE;
END_IF

// Loi khong doc duoc code may vision
T_Alarm[56]( IN := GVL.Pro4_.Auto.Alarm_Not_barcode_VS, PT := T#1S);
IF T_Alarm[56].Q THEN
	GVL.Alarm_P4.Read_Barcode_VS := TRUE;
ELSE
	GVL.Alarm_P4.Read_Barcode_VS := FALSE;
END_IF

// Loi day hang bang tai NG
T_Alarm[57]( IN:= NOT GVL.X[42] AND POU_MOTION.RUN_PROJECT, PT := T#5S);
IF T_Alarm[57].Q THEN
	GVL.Alarm_P4.Full_NG_CONV := TRUE;
ELSE
	GVL.Alarm_P4.Full_NG_CONV := FALSE;
END_IF
END_ACTION

ACTION Alarm_Robot:
// Loi Vacuum RB_A Tool 1
T_Alarm[0](IN:= ((GVL.RB_A_.Tool_1 AND NOT GVL.X[10]) OR (NOT GVL.RB_A_.Tool_1 AND GVL.X[10])) , PT := T#100MS);
IF T_Alarm[0].Q THEN 
	GVL.Alarm_Robot.A_Tool_1 := TRUE;
ELSE
	GVL.Alarm_Robot.A_Tool_1 := FALSE;
END_IF
// Loi Vacuum RB_A Tool 2
T_Alarm[1](IN:= ((GVL.RB_A_.Tool_2 AND NOT GVL.X[11]) OR (NOT GVL.RB_A_.Tool_2 AND GVL.X[11])) , PT := T#100MS); 
IF T_Alarm[1].Q THEN
	GVL.Alarm_Robot.A_Tool_2 := TRUE;
ELSE
	GVL.Alarm_Robot.A_Tool_2 := FALSE;
END_IF
// Loi Vacuum RB_B Tool 1
T_Alarm[2](IN:= ((GVL.RB_B_.Tool_1 AND NOT GVL.X[12]) OR (NOT GVL.RB_B_.Tool_1 AND GVL.X[12])) , PT := T#100MS); 
IF T_Alarm[2].Q THEN
	GVL.Alarm_Robot.B_Tool_1 := TRUE;
ELSE
	GVL.Alarm_Robot.B_Tool_1 := FALSE;
END_IF

// Loi Vacuum RB_B Tool 2
T_Alarm[3](IN:= ((GVL.RB_B_.Tool_2 AND NOT GVL.X[13]) OR (NOT GVL.RB_B_.Tool_2 AND GVL.X[13])) , PT := T#100MS); 
IF T_Alarm[3].Q THEN
	GVL.Alarm_Robot.B_Tool_2 := TRUE;
ELSE
	GVL.Alarm_Robot.B_Tool_2 := FALSE;
END_IF
END_ACTION

END_PROGRAM

// Just_Motion_Control_x86_64_Linux_SM_WV/Application/PRG_ROBOT/POU_TransFormOXYR
PROGRAM POU_TransFormOXYR
VAR
	P1_Old, P2_Old, P3_Old, P1_New, P2_New, P3_New: ST_POS;
	P_Pick_Old, P_Pick_New : ST_POS;
	Save_P1_Old, Save_P2_Old, Save_P3_Old, Save_P1_New, Save_P2_New, Save_P3_New, Cal_Transform, Cal_NewPoint, Save_P_Pick: BOOL;
	TF_Cal : ST_ScaraTransformDeg;
END_VAR

IF Save_P1_Old THEN
	GVL_1.DATA_RB_A.Data_Tranform[0].P1_Old.X := TO_REAL(GVL.RB_A_.CUR_X);
	GVL_1.DATA_RB_A.Data_Tranform[0].P1_Old.Y := TO_REAL(GVL.RB_A_.CUR_Y);
	GVL_1.DATA_RB_A.Data_Tranform[0].P1_Old.Z := TO_REAL(GVL.RB_A_.CUR_Z);
	GVL_1.DATA_RB_A.Data_Tranform[0].P1_Old.A := TO_REAL(GVL.RB_A_.CUR_R);
END_IF
IF Save_P2_Old THEN
	GVL_1.DATA_RB_A.Data_Tranform[0].P2_Old.X := TO_REAL(GVL.RB_A_.CUR_X);
	GVL_1.DATA_RB_A.Data_Tranform[0].P2_Old.Y := TO_REAL(GVL.RB_A_.CUR_Y);
	GVL_1.DATA_RB_A.Data_Tranform[0].P2_Old.Z := TO_REAL(GVL.RB_A_.CUR_Z);
	GVL_1.DATA_RB_A.Data_Tranform[0].P2_Old.A := TO_REAL(GVL.RB_A_.CUR_R);
END_IF
IF Save_P3_Old THEN
	GVL_1.DATA_RB_A.Data_Tranform[0].P3_Old.X := TO_REAL(GVL.RB_A_.CUR_X);
	GVL_1.DATA_RB_A.Data_Tranform[0].P3_Old.Y := TO_REAL(GVL.RB_A_.CUR_Y);
	GVL_1.DATA_RB_A.Data_Tranform[0].P3_Old.Z := TO_REAL(GVL.RB_A_.CUR_Z);
	GVL_1.DATA_RB_A.Data_Tranform[0].P3_Old.A := TO_REAL(GVL.RB_A_.CUR_R);
END_IF
IF Save_P1_New THEN
	GVL_1.DATA_RB_A.Data_Tranform[0].P1_New.X := TO_REAL(GVL.RB_A_.CUR_X);
	GVL_1.DATA_RB_A.Data_Tranform[0].P1_New.Y := TO_REAL(GVL.RB_A_.CUR_Y);
	GVL_1.DATA_RB_A.Data_Tranform[0].P1_New.Z := TO_REAL(GVL.RB_A_.CUR_Z);
	GVL_1.DATA_RB_A.Data_Tranform[0].P1_New.A := TO_REAL(GVL.RB_A_.CUR_R);
END_IF
IF Save_P2_New THEN
	GVL_1.DATA_RB_A.Data_Tranform[0].P2_New.X := TO_REAL(GVL.RB_A_.CUR_X);
	GVL_1.DATA_RB_A.Data_Tranform[0].P2_New.Y := TO_REAL(GVL.RB_A_.CUR_Y);
	GVL_1.DATA_RB_A.Data_Tranform[0].P2_New.Z := TO_REAL(GVL.RB_A_.CUR_Z);
	GVL_1.DATA_RB_A.Data_Tranform[0].P2_New.A := TO_REAL(GVL.RB_A_.CUR_R);
END_IF
IF Save_P3_New THEN
	GVL_1.DATA_RB_A.Data_Tranform[0].P3_New.X := TO_REAL(GVL.RB_A_.CUR_X);
	GVL_1.DATA_RB_A.Data_Tranform[0].P3_New.Y := TO_REAL(GVL.RB_A_.CUR_Y);
	GVL_1.DATA_RB_A.Data_Tranform[0].P3_New.Z := TO_REAL(GVL.RB_A_.CUR_Z);
	GVL_1.DATA_RB_A.Data_Tranform[0].P3_New.A := TO_REAL(GVL.RB_A_.CUR_R);
END_IF
IF Save_P_Pick THEN
	P_Pick_Old.X := TO_REAL(GVL.RB_B_.CUR_X);
	P_Pick_Old.Y := TO_REAL(GVL.RB_B_.CUR_Y);
	P_Pick_Old.Z := TO_REAL(GVL.RB_B_.CUR_Z);
	P_Pick_Old.A := TO_REAL(GVL.RB_B_.CUR_R);
END_IF
IF Cal_Transform THEN
	TF_Cal := CalcScaraTransformDeg(P1_old := GVL_1.DATA_RB_A.Data_Tranform[0].P1_old,
    P2_old := GVL_1.DATA_RB_A.Data_Tranform[0].P2_old,
    P3_old := GVL_1.DATA_RB_A.Data_Tranform[0].P3_old,
    P1_new := GVL_1.DATA_RB_A.Data_Tranform[0].P1_new,
    P2_new := GVL_1.DATA_RB_A.Data_Tranform[0].P2_new,
    P3_new := GVL_1.DATA_RB_A.Data_Tranform[0].P3_new,
    RefX := -1.0,
    RefY := 0,
    Eps := 0.000001);
END_IF
IF Cal_NewPoint THEN
	P_Pick_New := ApplyTransformOnePointDeg(Tf := TF_Cal,
        PointIn := P_Pick_Old
    );
END_IF

END_PROGRAM

// Just_Motion_Control_x86_64_Linux_SM_WV/Application/FC_/CalcScaraTransformDeg
FUNCTION CalcScaraTransformDeg  : ST_ScaraTransformDeg
VAR_INPUT
	P1_old : Pos_Coordsystem;
    P2_old : Pos_Coordsystem;
    P3_old : Pos_Coordsystem;

    P1_new : Pos_Coordsystem;
    P2_new : Pos_Coordsystem;
    P3_new : Pos_Coordsystem;

    RefX : LREAL;
    RefY : LREAL;

    Eps  : LREAL;
END_VAR
VAR
	Tf : ST_ScaraTransformDeg;

    vx_o, vy_o : LREAL;
    vx_n, vy_n : LREAL;
    len_o, len_n : LREAL;

    ux_o, uy_o : LREAL;
    ux_n, uy_n : LREAL;

    theta_o_rad, theta_n_rad : LREAL;
    theta_o_deg, theta_n_deg : LREAL;

    cross_o, cross_n : LREAL;
    dot_o, dot_n : LREAL;

    refLen : LREAL;
    refUx  : LREAL;
    refUy  : LREAL;
END_VAR

Tf.Valid := FALSE;
Tf.Error := FALSE;
Tf.ErrorID := 0;
Tf.CosT := 0.0;
Tf.SineT := 0.0;
Tf.ThetaDeg := 0.0;
Tf.Dx := 0.0;
Tf.Dy := 0.0;
Tf.Dz := 0.0;
Tf.DeltaR := 0.0;

refLen := SQRT(RefX*RefX + RefY*RefY);
IF refLen < Eps THEN
    Tf.Error := TRUE;
    Tf.ErrorID := 99;
    CalcScaraTransformDeg := Tf;
    RETURN;
END_IF;

refUx := RefX / refLen;
refUy := RefY / refLen;

// OLD Tinh vector P1_old-> P2_old
vx_o := P2_old.X - P1_old.X;
vy_o := P2_old.Y - P1_old.Y;
// Kiem tra neu toa do 2 diem qua gan nhau
len_o := SQRT(vx_o*vx_o + vy_o*vy_o);
IF len_o < Eps THEN
    Tf.Error := TRUE;
    Tf.ErrorID := 1; // Loi 2 diem trung nhau
    CalcScaraTransformDeg := Tf;
    RETURN;
END_IF;
// tinh vector theo don vi 1
ux_o := vx_o / len_o;
uy_o := vy_o / len_o;
// Kiem tra xem huong P1_0ld -> p2_old co bi nguoc hay khong
dot_o := ux_o*refUx + uy_o*refUy;
IF dot_o <= 0.0 THEN
    Tf.Error := TRUE;
    Tf.ErrorID := 2;
    CalcScaraTransformDeg := Tf;
    RETURN;
END_IF;

// Kiem tra P3 co dung huong khong
cross_o := vx_o*(P3_old.Y - P1_old.Y) - vy_o*(P3_old.X - P1_old.X);
IF cross_o <= Eps THEN
    Tf.Error := TRUE;
    Tf.ErrorID := 3;
    CalcScaraTransformDeg := Tf;
    RETURN;
END_IF;

//theta_o_rad := ATAN(vy_o/vx_o);
theta_o_rad := MyATAN2(vy_o,vx_o);
theta_o_deg := FC_Rad_To_Deg(theta_o_rad);

// NEW
vx_n := P2_new.X - P1_new.X;
vy_n := P2_new.Y - P1_new.Y;

len_n := SQRT(vx_n*vx_n + vy_n*vy_n);
IF len_n < Eps THEN
    Tf.Error := TRUE;
    Tf.ErrorID := 4;
    CalcScaraTransformDeg := Tf;
    RETURN;
END_IF;

ux_n := vx_n / len_n;
uy_n := vy_n / len_n;

dot_n := ux_n*refUx + uy_n*refUy;
IF dot_n <= 0.0 THEN
    Tf.Error := TRUE;
    Tf.ErrorID := 5;
    CalcScaraTransformDeg := Tf;
    //RETURN;
END_IF;

cross_n := vx_n*(P3_new.Y - P1_new.Y) - vy_n*(P3_new.X - P1_new.X);
IF cross_n <= Eps THEN
    Tf.Error := TRUE;
    Tf.ErrorID := 6;
    CalcScaraTransformDeg := Tf;
    RETURN;
END_IF;

theta_n_rad := MyATAN2(vy_n,vx_n);
theta_n_deg := FC_Rad_To_Deg(theta_n_rad);

// TRANSFORM
Tf.ThetaDeg := FC_NormalizeAngleDeg(theta_n_deg - theta_o_deg);
Tf.CosT := COS(FC_Deg_To_Rad(Tf.ThetaDeg));
Tf.SineT := SIN(FC_Deg_To_Rad(Tf.ThetaDeg));

Tf.Dx := P1_new.X - (P1_old.X*Tf.CosT - P1_old.Y*Tf.SineT);
Tf.Dy := P1_new.Y - (P1_old.X*Tf.SineT + P1_old.Y*Tf.CosT);
Tf.Dz := P1_new.Z - P1_old.Z;

Tf.DeltaR := FC_NormalizeAngleDeg(P1_new.A - (P1_old.A + Tf.ThetaDeg));

Tf.Valid := TRUE;
Tf.Error := FALSE;
Tf.ErrorID := 0;

CalcScaraTransformDeg := Tf;

END_FUNCTION

// Just_Motion_Control_x86_64_Linux_SM_WV/Application/FC_/MyATAN2
FUNCTION MyATAN2 : LREAL
VAR_INPUT
	y : LREAL;
    x : LREAL;
END_VAR
VAR
	pi : LREAL := 3.14159265358979;
END_VAR

IF x > 0 THEN
    MyATAN2 := ATAN(y / x);

ELSIF x < 0 AND y >= 0 THEN
    MyATAN2 := ATAN(y / x) + pi;

ELSIF x < 0 AND y < 0 THEN
    MyATAN2 := ATAN(y / x) - pi;

ELSIF x = 0 AND y > 0 THEN
    MyATAN2 := pi / 2.0;

ELSIF x = 0 AND y < 0 THEN
    MyATAN2 := -pi / 2.0;

ELSE
    MyATAN2 := 0.0;
END_IF;

END_FUNCTION

// Just_Motion_Control_x86_64_Linux_SM_WV/Application/FC_/FC_Rad_To_Deg
FUNCTION FC_Rad_To_Deg : LREAL
VAR_INPUT
	AngleRad : LREAL;
END_VAR
VAR
END_VAR

FC_Rad_To_Deg := AngleRad * 180.0 / 3.14159265358979;

END_FUNCTION

// Just_Motion_Control_x86_64_Linux_SM_WV/Application/FC_/FC_NormalizeAngleDeg
FUNCTION FC_NormalizeAngleDeg : LREAL
VAR_INPUT
    AngleDeg : LREAL;
END_VAR
VAR
    A : LREAL;
END_VAR

A := AngleDeg;

WHILE A > 180.0 DO
    A := A - 360.0;
END_WHILE;

WHILE A < -180.0 DO
    A := A + 360.0;
END_WHILE;

FC_NormalizeAngleDeg := A;

END_FUNCTION

// Just_Motion_Control_x86_64_Linux_SM_WV/Application/FC_/FC_Deg_To_Rad
FUNCTION FC_Deg_To_Rad : LREAL
VAR_INPUT
	AngleDeg : LREAL;
END_VAR
VAR
END_VAR

FC_Deg_To_Rad := AngleDeg * 3.14159265358979 / 180.0;

END_FUNCTION

// Just_Motion_Control_x86_64_Linux_SM_WV/Application/FC_/ApplyTransformOnePointDeg
FUNCTION ApplyTransformOnePointDeg : ST_POS
VAR_INPUT
	 Tf      : ST_ScaraTransformDeg;
    PointIn : ST_POS;
END_VAR
VAR
	P : ST_POS;
END_VAR

P.X := PointIn.X * Tf.CosT - PointIn.Y * Tf.SineT + Tf.Dx;
P.Y := PointIn.X * Tf.SineT + PointIn.Y * Tf.CosT + Tf.Dy;
P.Z := PointIn.Z + Tf.Dz;
P.A := FC_NormalizeAngleDeg(PointIn.A + Tf.ThetaDeg + Tf.DeltaR);

ApplyTransformOnePointDeg := P;

END_FUNCTION

// Just_Motion_Control_x86_64_Linux_SM_WV/Application/PRG_ROBOT/POU_Main
PROGRAM POU_Main
VAR
    rTrig_Auto   : R_TRIG;
    rTrig_Manual : R_TRIG;
    rTrig_Lock   : R_TRIG;
	rTrig_B_Auto   : R_TRIG;
    rTrig_B_Manual : R_TRIG;
    rTrig_B_Lock   : R_TRIG;
	
	filedata : FB_FileManager;
	tsave, tload : TON;
	
	trigSave, TrigLoad : R_TRIG;
END_VAR

VAR
	//Input
	In_Start  : BOOL;
	In_Reset  : BOOL;
	In_Stop  : BOOL;
	In_EMG : BOOL;
	// Output
	Out_Red_Towerlamp : BOOL;
	Out_Yellow_Towerlamp  : BOOL;
	Out_Green_Towerlamp  : BOOL;
	Out_Buzz  : BOOL;
	
	Pulse_1s : BOOL;
	T_1s : TON;
	RunTime_s  : UDINT;   // Thời gian chạy (giây)
    StopTime_s : UDINT;   // Thời gian dừng
    WaitTime_s : UDINT;   // Thời gian chờ
    TotalTime_s: UDINT;   // Tổng thời gian
	
END_VAR


VAR
	// IN
	
	T_RESET_TS, T_RESET_VS,
	 T_OUT_RESET_TS, T_OUT_RESET_VS : TON;
	 First_Scan: BOOL := FALSE;
	 Read_Model_BF : BOOL;
END_VAR
VAR
    rSave_RB_A : R_TRIG;
    rLoad_RB_A : R_TRIG;
	rSave_RB_B : R_TRIG;
    rLoad_RB_B : R_TRIG;
	rSave_DT_Pro4 : R_TRIG;
    rLoad_DT_Pro4 : R_TRIG;
	rSave_DT_Pro4_Auto : R_TRIG;
    rLoad_DT_Pro4_Auto, rReadModel_BF : R_TRIG;
END_VAR

VAR
	i_1, i_cam : INT;
	S_fileName_Model : STRING;
	S_Robot_A_Name : STRING := 'file_data_RB_A_Project_';
	S_Robot_B_Name : STRING := 'file_data_RB_B_Project_';
	S_Robot_Name : STRING := 'file_data_RB_Project_';
	S_Robot_A_Name_Full : STRING := '';
	S_Robot_B_Name_Full : STRING := '';
	S_Robot_Name_Full : STRING := '';
	S_Model_No : STRING;
	rSave_Model : R_TRIG;
    rCall_Model : R_TRIG;
	
	r_Save_ToolConfig, r_Read_ToolConfig: R_TRIG;
	r_Save_ConveyorConfig,r_Read_ConveyorConfig: R_TRIG;
	r_Save_TrackingConfig, r_Read_TrackingConfig: R_TRIG;
	Read_Config_First : BOOL;
END_VAR

// update out - namnv

// namnv3103
IF NOT First_Scan THEN
	Read_Config_First := TRUE;
	Read_Model_BF := TRUE;
	First_Scan := TRUE;
	FOR i_cam := 0 TO 10 BY 1 DO
		GVL.Load_Data_Cam[i_cam] := TRUE;
	END_FOR
END_IF


// Call PG
ACT_StatusMode();
ACT_Out();
ACT_IN();
TimeTable();
ACT_SAVE_FILE();
ACT_SelectProjectRun();

ACTION ACT_IN:
// Bao gom input cua chung cua robot va dat ten rieng cho tung project
// Share robot
// update in
GVL.RB_Signal_In.HMI_START := GVL.X[6];
GVL.RB_Signal_In.HMI_RESET := GVL.X[8];
GVL.RB_Signal_In.HMI_EMG  := GVL.X[9];
GVL.RB_Signal_In.HMI_STOP   := GVL.X[7];
// Tool robot'
GVL.RB_Signal_In.SS_RBA_Tool_1( IN:= GVL.X[10], PT := T#10MS, Q =>);

GVL.RB_Signal_In.SS_RBA_Tool_2( IN:= GVL.X[11], PT := T#50MS, Q =>);

GVL.RB_Signal_In.SS_RBB_Tool_1( IN:= GVL.X[12], PT := T#50MS, Q =>);

GVL.RB_Signal_In.SS_RBB_Tool_2( IN:= GVL.X[13], PT := T#50MS, Q =>);


// Project 3
IF GVL.ProjectAndModel.Project_No_Current = 3 THEN	
	// Test sóng
	
